(* CODESYS project railCtrl1023.project

Project tree, tasks and I/O mapping:
  Device : CODESYS SoftMotion Win V3, 3S - Smart Software Solutions GmbH, order no. 309021, version 3.5.10.0
    application Application
      libraries: Standard, * (System); VisuDialogs, * (System)
      task MainTask (cyclic, interval 4 ms, priority 1) calls PLC_PRG, floorRailInterface, yysInterface
      task VISU_TASK (cyclic, interval 100 ms, priority 31) calls VisuElems.Visu_Prg
      program PLC_PRG [ST]
      floor_rail/
        program floorRailInterface [ST]: floorRailInterface_Status, floorRailInterface_Cmd
        struct_floor_rail/
          data type OilBlockUnit_Base
          data type OilBlockUnit_Status
          data type OilBlockUnit_Cmd
          data type OilBlockUnit_Status_Loc
          data type OilBlockUnit_Status_PosVal
          data type RatioValveD1
          data type RatioValveD2
          data type RatioValveD4
          data type RatioValveD3
          data type RatioValveD5
          data type RatioValveD6
          data type RatioValveD7
          UICell/
            data type UICell_OilBlock_Info
            data type UICell_OilBlock_Button
            data type UICell_RVD3
            data type UICell_RVD1
            data type UICell_RVD2
            data type UICell_RVD5
            data type UICell_RVD4
            data type UICell_RVD6
            data type UICell_RVD7
            data type UICell_OilBlock_Module
            data type UICell_OilBlock_Module_Info
            data type UICell_OilBlock_Module_Button
          data type propValve_Struct
        text list TextList
      ceiling_rail/
        struct_ceiling_rail/
      yy_station/
        struct_yystation/
          data type YyStation_Cmd
          data type YyStation_Status
          data type YyStation
        program yysInterface [ST]: yysInterface_Status, yysInterface_Cmd
      can/
        function swmc_C00_Rx [ST]
        struct_can/
          data type Can_baseframe
          data type Can_BUS_8Inputs
          data type Can_BUS_8Outputs
          data type Can_Bus_RXMsg_Buff
          data type Can_Bus_TXMsg_Buff
        function swmc_C00_Tx [ST]
        function CAN_Send_Data_SWMC [ST]
        function swmc_C01_Rx [ST]
        function swmc_C01_Tx [ST]
        function swmc_C02_Rx [ST]
        function swmc_C02_Tx [ST]
        function swmc_C09_Rx [ST]
        function swmc_C10_Rx [ST]
      global variables gImple
      global variables gUI
      global variables gCan
      display/
        visualisation YY_Station_Display
        Orig/
          visualisation Floor_Rail1
          Module/
            visualisation OilBlock_PrimButton
            visualisation OilBlock_PrimInfo
            visualisation ModuleX2
            visualisation ModuleX1
            visualisation ModuleX3
            visualisation ModuleX8
            visualisation ModuleX4
            visualisation ModuleX5
            visualisation ModuleDTD
          visualisation Floor_Rail2
          visualisation Floor_Rail_345
          visualisation Floor_Rail6
          visualisation Floor_Rail7
          visualisation Floor_Rail_12
        visualisation Floor_Rail
        visualisation main_UI
    SoftMotion General Axis Pool
  libraries: VisuSymbols, 3.5.10.0 (System)
  text list GlobalTextList
*)

// Device/Application/yy_station/struct_yystation/YyStation_Cmd
TYPE YyStation_Cmd :
STRUCT
	InverterFan_Ctrl  		:BOOL;   //变频风机控制 0x400-1.0
	OilPumpFan_Ctrl   		:BOOL;   //油泵风机控制 0x400-1.1
	//------以下变量暂未使用,取自水平库-----------------------------------
	OilPumpMotor_Ctrl 		:BOOL;   //油泵电机控制
	OilPumpMotor_PN_Ctrl 	:BOOL;   //油泵电机正反转控制
	HL_Mode_Ctrl 			:BOOL;   //高低速模式
	KEEP_Mode_Ctrl          :BOOL;   //恒速模式
	Energy_Swith			:BOOL;   //储能控制
	Oil_Pre_Val             :WORD;   //油压控制
END_STRUCT
END_TYPE

// Device/Application/yy_station/struct_yystation/YyStation_Status
TYPE YyStation_Status :
STRUCT

	pressureStatus					: REAL;		//压力开关S1|0x300-Byt1~2
	temperatureStatus				: REAL;		//温度开关S14|0x300-Byt3~4
	yeweiStatus						: BOOL;		//液位开关S15|0x300-Byt5~6

	FrequencyConversion_Fault 		: BOOL;			//变频故障|0x300-7.0
	FrequencyConversion_Run 		: BOOL;			//变频运行|0x300-7.1
	HydraulicStation_Power			: BOOL;			//液压站上电-状态|0x300-7.2
	Control_Power					: BOOL;			//控制总电源上电状态|0x300-7.3
	InverterFan_Run 				: BOOL;			//变频风机运行状态|0x300-7.4
	OilPumpFan						: BOOL;			//冷却油泵状态|0x300-7.5
	OilPumpM_Fault 					: BOOL;			//油泵电机故障状态|0x300-7.6
	InverterFan_Fault 				: BOOL;			//变频风机故障|0x300-7.7
	
	//地轨部分压力传感器
	pressureV2						: REAL;			//压力传感器S2P|0x316-Byt1~2
	pressureV3						: REAL;			//压力传感器S3P|0x316-Byt3~4
	pressureV4						: REAL;			//压力传感器S4P|0x326-Byt1~2
	pressureV5						: REAL;			//压力传感器S5P|0x326-Byt3~4
	//天轨部分压力传感器
	pressureV8						: REAL;			//压力传感器S8P|0x356-Byt1~2
	pressureV9						: REAL;			//压力传感器S9P|0x356-Byt3~4
	pressureV10						: REAL;			//压力传感器S10P|0x366-Byt1~2
	pressureV11						: REAL;			//压力传感器S11P|0x366-Byt3~4
	

	

END_STRUCT
END_TYPE

// Device/Application/yy_station/struct_yystation/YyStation
TYPE YyStation :
STRUCT
	Cmd		:YyStation_Cmd;		//液压站指令
	Status	:YyStation_Status;	//液压站状态
	
END_STRUCT
END_TYPE

// Device/Application/can/struct_can/Can_baseframe
TYPE Can_baseframe :
STRUCT
	id		: UINT;
	data	: ARRAY[1..8] OF BYTE;
END_STRUCT
END_TYPE

// Device/Application/can/struct_can/Can_BUS_8Inputs
TYPE Can_BUS_8Inputs :          //输入缓存结构 EL6751-8Message_IN
STRUCT
	TxCounter			: UINT;
	RxCounter			: UINT;
	NoOfRxMessages 	 	: UINT;
	TransactionNumber	: UINT;
	RXMsg				: ARRAY[1..8] OF Can_Bus_RXMsg_Buff;
	CAN_State			: UINT;
	Align				: UINT;
	RX_Error_Cnt		: BYTE;
	TX_Error_Cnt		: BYTE;
END_STRUCT
END_TYPE

// Device/Application/can/struct_can/Can_BUS_8Outputs
TYPE Can_BUS_8Outputs :		//输出缓存结构 EL6751-8Message_OUT
STRUCT
	TxCounter		: UINT;
	RxCounter		: UINT;
	NoOfTxMessages 	: UINT;
	TXMsg			: ARRAY[1..8] OF Can_Bus_TXMsg_Buff;
	CAN_Control		: UINT;
END_STRUCT
END_TYPE

// Device/Application/can/struct_can/Can_Bus_RXMsg_Buff
TYPE Can_Bus_RXMsg_Buff:
STRUCT
	RxMsg_CobId		: UINT;
	RxMsg_Byte  	: ARRAY[1..8] OF BYTE;
END_STRUCT
END_TYPE

// Device/Application/can/struct_can/Can_Bus_TXMsg_Buff
TYPE Can_Bus_TXMsg_Buff :
STRUCT
	TxMsg_TransactionNumber		: UINT;
	TxMsg_CobId					: UINT;
	TxMsg_Byte  				: ARRAY[1..8] OF BYTE;
END_STRUCT
END_TYPE

// Device/Application/floor_rail/struct_floor_rail/OilBlockUnit_Base
TYPE OilBlockUnit_Base :
STRUCT
	cmd		:OilBlockUnit_Cmd;				//发送油缸指令
	status	:OilBlockUnit_Status;			//油缸状态
	cnt     :UINT;			  				//超时计数

END_STRUCT
END_TYPE

// Device/Application/floor_rail/struct_floor_rail/OilBlockUnit_Status
TYPE OilBlockUnit_Status :
STRUCT
	
	posVal			:OilBlockUnit_Status_PosVal;	//传感器位置值
	locStat			:OilBlockUnit_Status_Loc;		//位置状态
	
END_STRUCT
END_TYPE

// Device/Application/floor_rail/struct_floor_rail/OilBlockUnit_Cmd
TYPE OilBlockUnit_Cmd :
STRUCT
	E_Open	:BOOL;
	R_Open 	:BOOL;
END_STRUCT
END_TYPE

// Device/Application/floor_rail/struct_floor_rail/OilBlockUnit_Status_Loc
{attribute 'qualified_only'}
{attribute 'strict'}
TYPE OilBlockUnit_Status_Loc :
(
	enum_Run  		:= 0,   //运行中
	enum_Extend 	:= 1,	//伸出完成
	enum_Retract  	:= 2,	//缩回完成

	enum_Err  		:= 10   //错误
);
END_TYPE

// Device/Application/floor_rail/struct_floor_rail/OilBlockUnit_Status_PosVal
TYPE OilBlockUnit_Status_PosVal :
STRUCT
	Extend 		:REAL;    //伸出位置
	Retract   	:REAL;    //收回位置
	Current 	:REAL;    //当前位置
END_STRUCT
END_TYPE

// Device/Application/floor_rail/struct_floor_rail/RatioValveD1
TYPE RatioValveD1 :
STRUCT
	percenVal	: WORD;              				//比例阀DTD1|0x410-Byt1~2 0-65535 对应 0-100
	
	RVD1		:ARRAY[1..12] OF OilBlockUnit_Base;
	
	D00Q1	 	: OilBlockUnit_Base;				//DTD1连接的油缸
	D00Q2	 	: OilBlockUnit_Base;				//DTD1连接的油缸
	
	D28L1	 	: OilBlockUnit_Base;				//DTD1连接的油缸
	D28L2	 	: OilBlockUnit_Base;				//DTD1连接的油缸
	
	D29L	 	: OilBlockUnit_Base;				//DTD1连接的油缸
	D30L	 	: OilBlockUnit_Base;				//DTD1连接的油缸	

	D00L1	 	: OilBlockUnit_Base;				//DTD1连接的油缸
	D00L2	 	: OilBlockUnit_Base;				//DTD1连接的油缸
	
	D01L	 	: OilBlockUnit_Base;				//DTD1连接的油缸
	
	D28Q	 	: OilBlockUnit_Base;				//DTD1连接的油缸
	D29Q	 	: OilBlockUnit_Base;				//DTD1连接的油缸
		
	D30Q	 	: OilBlockUnit_Base;				//DTD1连接的油缸
	
	END_STRUCT
END_TYPE

// Device/Application/floor_rail/struct_floor_rail/RatioValveD2
TYPE RatioValveD2 :
STRUCT
	percenVal	: WORD;              				//比例阀DTD2|0x410-Byt3~4 0-65535 对应 0-100
	
	RVD2		:ARRAY[1..11] OF OilBlockUnit_Base;
	
	D02L	 	: OilBlockUnit_Base;				//DTD2连接的油缸
	D03L	 	: OilBlockUnit_Base;				//DTD2连接的油缸
	D04L	 	: OilBlockUnit_Base;				//DTD2连接的油缸
	
	D05L	 	: OilBlockUnit_Base;				//DTD2连接的油缸
	
	D06L	 	: OilBlockUnit_Base;				//DTD2连接的油缸
	D07L	 	: OilBlockUnit_Base;				//DTD2连接的油缸
	D08L	 	: OilBlockUnit_Base;				//DTD2连接的油缸
	
	D09L	 	: OilBlockUnit_Base;				//DTD2连接的油缸
	
	D10L	 	: OilBlockUnit_Base;				//DTD2连接的油缸
	D11L	 	: OilBlockUnit_Base;				//DTD2连接的油缸
	D12L	 	: OilBlockUnit_Base;				//DTD2连接的油缸

END_STRUCT
END_TYPE

// Device/Application/floor_rail/struct_floor_rail/RatioValveD4
TYPE RatioValveD4 :
STRUCT
	percenVal	: WORD;              				//比例阀DTD3|0x410-Byt5~6 0-65535 对应 0-100
	
	RVD4		:ARRAY[1..8] OF OilBlockUnit_Base;
	
	D05Q1	 	: OilBlockUnit_Base;				//DTD3连接的油缸
	D05Q2	 	: OilBlockUnit_Base;				//DTD3连接的油缸
	D06Q1	 	: OilBlockUnit_Base;				//DTD3连接的油缸
	D06Q2	 	: OilBlockUnit_Base;				//DTD3连接的油缸
	D07Q1	 	: OilBlockUnit_Base;				//DTD3连接的油缸
	D07Q2	 	: OilBlockUnit_Base;				//DTD3连接的油缸
	D08Q1	 	: OilBlockUnit_Base;				//DTD3连接的油缸
	D08Q2	 	: OilBlockUnit_Base;				//DTD3连接的油缸
END_STRUCT
END_TYPE

// Device/Application/floor_rail/struct_floor_rail/RatioValveD3
TYPE RatioValveD3 :
STRUCT
	percenVal	: WORD;              				//比例阀DTD4|0x410-Byt7~8 0-65535 对应 0-100
	
	RVD3		:ARRAY[1..8] OF OilBlockUnit_Base;
	
	D01Q1	 	: OilBlockUnit_Base;				//DTD4连接的油缸
	D01Q2	 	: OilBlockUnit_Base;				//DTD4连接的油缸
	D02Q1	 	: OilBlockUnit_Base;				//DTD4连接的油缸
	D02Q2	 	: OilBlockUnit_Base;				//DTD4连接的油缸	
	D03Q1	 	: OilBlockUnit_Base;				//DTD4连接的油缸
	D03Q2	 	: OilBlockUnit_Base;				//DTD4连接的油缸
	D04Q1	 	: OilBlockUnit_Base;				//DTD4连接的油缸
	D04Q2	 	: OilBlockUnit_Base;				//DTD4连接的油缸
END_STRUCT
END_TYPE

// Device/Application/floor_rail/struct_floor_rail/RatioValveD5
TYPE RatioValveD5 :
STRUCT
	percenVal	: WORD;              				//比例阀DTD5|0x411-Byt1~2 0-65535 对应 0-100
	
	RVD5		:ARRAY[1..8] OF OilBlockUnit_Base;
	
	D09Q1	 	: OilBlockUnit_Base;				//DTD5连接的油缸
	D09Q2	 	: OilBlockUnit_Base;				//DTD5连接的油缸
	D10Q1	 	: OilBlockUnit_Base;				//DTD5连接的油缸
	D10Q2	 	: OilBlockUnit_Base;				//DTD5连接的油缸
	D11Q1	 	: OilBlockUnit_Base;				//DTD5连接的油缸
	D11Q2	 	: OilBlockUnit_Base;				//DTD5连接的油缸	
	D12Q1	 	: OilBlockUnit_Base;				//DTD5连接的油缸
	D12Q2	 	: OilBlockUnit_Base;				//DTD5连接的油缸
END_STRUCT
END_TYPE

// Device/Application/floor_rail/struct_floor_rail/RatioValveD6
TYPE RatioValveD6 :
STRUCT
	percenVal	: WORD;              				//比例阀DTD6|0x420-Byt1~2 0-65535 对应 0-100
	
	RVD6		:ARRAY[1..8] OF OilBlockUnit_Base;
	
	D13Q	 	: OilBlockUnit_Base;				//DTD6连接的油缸
	D13L	 	: OilBlockUnit_Base;				//DTD6连接的油缸
	D14Q	 	: OilBlockUnit_Base;				//DTD6连接的油缸
	D14L	 	: OilBlockUnit_Base;				//DTD6连接的油缸
	D15Q	 	: OilBlockUnit_Base;				//DTD6连接的油缸
	D15L	 	: OilBlockUnit_Base;				//DTD6连接的油缸
	D16L1	 	: OilBlockUnit_Base;				//DTD6连接的油缸
	D16L2	 	: OilBlockUnit_Base;				//DTD6连接的油缸

END_STRUCT
END_TYPE

// Device/Application/floor_rail/struct_floor_rail/RatioValveD7
TYPE RatioValveD7 :
STRUCT
	percenVal	: WORD;              				//比例阀DTD7|0x420-Byt3~4 0-65535 对应 0-100
	
	RVD7		:ARRAY[1..23] OF OilBlockUnit_Base;
	
	D17Q	 	: OilBlockUnit_Base;				//DTD7连接的油缸
	D17L1	 	: OilBlockUnit_Base;				//DTD7连接的油缸
	D17L2	 	: OilBlockUnit_Base;				//DTD7连接的油缸
	D18Q	 	: OilBlockUnit_Base;				//DTD7连接的油缸
	D18L	 	: OilBlockUnit_Base;				//DTD7连接的油缸
	D19Q	 	: OilBlockUnit_Base;				//DTD7连接的油缸
	D19L	 	: OilBlockUnit_Base;				//DTD7连接的油缸
	D20Q	 	: OilBlockUnit_Base;				//DTD7连接的油缸
	D20L	 	: OilBlockUnit_Base;				//DTD7连接的油缸
	D21Q	 	: OilBlockUnit_Base;				//DTD7连接的油缸
	D21L	 	: OilBlockUnit_Base;				//DTD7连接的油缸
	D22Q	 	: OilBlockUnit_Base;				//DTD7连接的油缸
	D22L	 	: OilBlockUnit_Base;				//DTD7连接的油缸
	D23Q	 	: OilBlockUnit_Base;				//DTD7连接的油缸
	D23L	 	: OilBlockUnit_Base;				//DTD7连接的油缸
	D24Q	 	: OilBlockUnit_Base;				//DTD7连接的油缸
	D24L	 	: OilBlockUnit_Base;				//DTD7连接的油缸
	D25Q	 	: OilBlockUnit_Base;				//DTD7连接的油缸
	D25L	 	: OilBlockUnit_Base;				//DTD7连接的油缸
	D26Q	 	: OilBlockUnit_Base;				//DTD7连接的油缸
	D26L	 	: OilBlockUnit_Base;				//DTD7连接的油缸
	D27L1	 	: OilBlockUnit_Base;				//DTD7连接的油缸
	D27L2	 	: OilBlockUnit_Base;				//DTD7连接的油缸



END_STRUCT
END_TYPE

// Device/Application/floor_rail/struct_floor_rail/UICell/UICell_OilBlock_Info
TYPE UICell_OilBlock_Info :
STRUCT
	strName			:STRING;
	rPosition		:REAL;
	rPercent		:REAL;
END_STRUCT
END_TYPE

// Device/Application/floor_rail/struct_floor_rail/UICell/UICell_OilBlock_Button
TYPE UICell_OilBlock_Button :
STRUCT
	bExtend			: BOOL;	
	bRetract		: BOOL;
	bStop			: BOOL;
END_STRUCT
END_TYPE

// Device/Application/floor_rail/struct_floor_rail/UICell/UICell_RVD3
TYPE UICell_RVD3 :
STRUCT
	bRVD3_enable	:BOOL;
	rRVD3Percent	:REAL;
	S1		:UICell_OilBlock_Button;
	D01Q1	:UICell_OilBlock_Info;
	D01Q2	:UICell_OilBlock_Info;
	D02Q1	:UICell_OilBlock_Info;
	D02Q2	:UICell_OilBlock_Info;
	
	D03Q1	:UICell_OilBlock_Info;
	D03Q2	:UICell_OilBlock_Info;
	D04Q1	:UICell_OilBlock_Info;
	D04Q2	:UICell_OilBlock_Info;

END_STRUCT
END_TYPE

// Device/Application/floor_rail/struct_floor_rail/UICell/UICell_RVD1
TYPE UICell_RVD1 :
STRUCT
	
	bRVD1_enable	:BOOL;
	rRVD1Percent	:REAL;

	S1		:UICell_OilBlock_Button;
	D00Q1	:UICell_OilBlock_Info;
	D00Q2	:UICell_OilBlock_Info;
	
	
	S2		:UICell_OilBlock_Button;
	D28L1	:UICell_OilBlock_Info;
	D28L2	:UICell_OilBlock_Info;
	
	S3		:UICell_OilBlock_Button;
	D29L	:UICell_OilBlock_Info;
	D30L	:UICell_OilBlock_Info;
	
	S4		:UICell_OilBlock_Button;
	D00L1	:UICell_OilBlock_Info;
	D00L2	:UICell_OilBlock_Info;
	
	S5		:UICell_OilBlock_Button;
	D01L	:UICell_OilBlock_Info;

	S6		:UICell_OilBlock_Button;
	D28Q	:UICell_OilBlock_Info;
	D29Q	:UICell_OilBlock_Info;
	
	S7		:UICell_OilBlock_Button;
	D30Q	:UICell_OilBlock_Info;

END_STRUCT
END_TYPE

// Device/Application/floor_rail/struct_floor_rail/UICell/UICell_RVD2
TYPE UICell_RVD2 :
STRUCT
	
	bRVD2_enable	:BOOL;
	rRVD2Percent	:REAL;
	
	S1		:UICell_OilBlock_Button;
	D02L	:UICell_OilBlock_Info;
	D03L	:UICell_OilBlock_Info;
	D04L	:UICell_OilBlock_Info;
	
	S2		:UICell_OilBlock_Button;
	D05L	:UICell_OilBlock_Info;
	
	S3		:UICell_OilBlock_Button;
	D06L	:UICell_OilBlock_Info;
	D07L	:UICell_OilBlock_Info;
	D08L	:UICell_OilBlock_Info;
	
	S4		:UICell_OilBlock_Button;
	D09L	:UICell_OilBlock_Info;

	S5		:UICell_OilBlock_Button;
	D10L	:UICell_OilBlock_Info;
	D11L	:UICell_OilBlock_Info;
	D12L	:UICell_OilBlock_Info;

END_STRUCT
END_TYPE

// Device/Application/floor_rail/struct_floor_rail/UICell/UICell_RVD5
TYPE UICell_RVD5 :
STRUCT
	bRVD5_enable	:BOOL;
	rRVD5Percent	:REAL;
	S1		:UICell_OilBlock_Button;
	D09Q1	:UICell_OilBlock_Info;
	D09Q2	:UICell_OilBlock_Info;
	D10Q1	:UICell_OilBlock_Info;
	D10Q2	:UICell_OilBlock_Info;
	
	D11Q1	:UICell_OilBlock_Info;
	D11Q2	:UICell_OilBlock_Info;
	D12Q1	:UICell_OilBlock_Info;
	D12Q2	:UICell_OilBlock_Info;

END_STRUCT
END_TYPE

// Device/Application/floor_rail/struct_floor_rail/UICell/UICell_RVD4
TYPE UICell_RVD4 :
STRUCT
	bRVD4_enable	:BOOL;
	rRVD4Percent	:REAL;
	S1		:UICell_OilBlock_Button;
	D05Q1	:UICell_OilBlock_Info;
	D05Q2	:UICell_OilBlock_Info;
	D06Q1	:UICell_OilBlock_Info;
	D06Q2	:UICell_OilBlock_Info;

	D07Q1	:UICell_OilBlock_Info;
	D07Q2	:UICell_OilBlock_Info;
	D08Q1	:UICell_OilBlock_Info;
	D08Q2	:UICell_OilBlock_Info;

END_STRUCT
END_TYPE

// Device/Application/floor_rail/struct_floor_rail/UICell/UICell_RVD6
TYPE UICell_RVD6 :
STRUCT
	bRVD6_enable	:BOOL;
	rRVD6Percent	:REAL;
	S1		:UICell_OilBlock_Button;
	D13Q	:UICell_OilBlock_Info;
	D14Q	:UICell_OilBlock_Info;
		
	S2		:UICell_OilBlock_Button;
	D15Q	:UICell_OilBlock_Info;
	
	S3		:UICell_OilBlock_Button;
	D13L	:UICell_OilBlock_Info;
	D14L	:UICell_OilBlock_Info;
	
	S4		:UICell_OilBlock_Button;
	D15L	:UICell_OilBlock_Info;

	S5		:UICell_OilBlock_Button;
	D16L1	:UICell_OilBlock_Info;
	D16L2	:UICell_OilBlock_Info;


END_STRUCT
END_TYPE

// Device/Application/floor_rail/struct_floor_rail/UICell/UICell_RVD7
TYPE UICell_RVD7 :
STRUCT
	bRVD7_enable	:BOOL;
	rRVD7Percent	:REAL;
	
	S1		:UICell_OilBlock_Button;
	D18L	:UICell_OilBlock_Info;
	D19L	:UICell_OilBlock_Info;
	D20L	:UICell_OilBlock_Info;
	D21L	:UICell_OilBlock_Info;
		
	S2		:UICell_OilBlock_Button;
	D22L	:UICell_OilBlock_Info;
	
	S3		:UICell_OilBlock_Button;
	D23L	:UICell_OilBlock_Info;
	D24L	:UICell_OilBlock_Info;
	D25L	:UICell_OilBlock_Info;
	D26L	:UICell_OilBlock_Info;
	
	S4		:UICell_OilBlock_Button;
	D17Q	:UICell_OilBlock_Info;
	D18Q	:UICell_OilBlock_Info;
	D19Q	:UICell_OilBlock_Info;
	D20Q	:UICell_OilBlock_Info;
	D21Q	:UICell_OilBlock_Info;

	S5		:UICell_OilBlock_Button;
	D22Q	:UICell_OilBlock_Info;
	D23Q	:UICell_OilBlock_Info;
	D24Q	:UICell_OilBlock_Info;
	D25Q	:UICell_OilBlock_Info;
	D26Q	:UICell_OilBlock_Info;
	
	S6		:UICell_OilBlock_Button;
	D17L1	:UICell_OilBlock_Info;
	D17L2	:UICell_OilBlock_Info;
	
	S7		:UICell_OilBlock_Button;
	D27L1	:UICell_OilBlock_Info;
	D27L2	:UICell_OilBlock_Info;

END_STRUCT
END_TYPE

// Device/Application/floor_rail/struct_floor_rail/propValve_Struct
TYPE propValve_Struct :
STRUCT
	D1	:RatioValveD1;
	D2	:RatioValveD2;
	D3	:RatioValveD3;
	D4	:RatioValveD4;
	D5	:RatioValveD5;
	D6	:RatioValveD6;
	D7	:RatioValveD7;

	
END_STRUCT
END_TYPE

// Device/Application/floor_rail/struct_floor_rail/UICell/UICell_OilBlock_Module
TYPE UICell_OilBlock_Module :
STRUCT
	
	sColumn				:ARRAY[1..8] OF UICell_OilBlock_Module_Button;
	sRow				:ARRAY[1..8] OF UICell_OilBlock_Module_Info;

END_STRUCT
END_TYPE

// Device/Application/floor_rail/struct_floor_rail/UICell/UICell_OilBlock_Module_Info
TYPE UICell_OilBlock_Module_Info :
STRUCT
	strName			:STRING;
	rPosition		:REAL;
	rPercent		:REAL;
END_STRUCT
END_TYPE

// Device/Application/floor_rail/struct_floor_rail/UICell/UICell_OilBlock_Module_Button
TYPE UICell_OilBlock_Module_Button :
STRUCT
	bExtend			: BOOL;	
	bRetract		: BOOL;
	bStop			: BOOL;
END_STRUCT
END_TYPE

// Device/Application/gImple
{attribute 'qualified_only'}
VAR_GLOBAL
	





	hydraPresStation	:YyStation;
	propValve			:propValve_Struct;
	
	
	
END_VAR

// Device/Application/gUI
{attribute 'qualified_only'}
VAR_GLOBAL
	
//液压站部分
	//压力
	rPressureVal1				:REAL;			//压力传感器SQ1P(压力开关S1)
	rPressureVal2				:REAL;			//压力传感器SQ2P
	rPressureVal3				:REAL;			//压力传感器SQ3P
	rPressureVal4				:REAL;			//压力传感器SQ4P
	rPressureVal5				:REAL;			//压力传感器SQ5P	
	//状态
	rTemperature				:REAL;			//温度值
	bFluidLevel					:BOOL;			//液位值
	
	bYysPower	 		 		:BOOL;			//液压站上电
	bCtrlPower	  		 		:BOOL;			//控制电源上电
	bFreqConverterFan			:BOOL;    	    //变频风机启动
	bFreqConverter				:BOOL;			//变频器运行
	
	bOilPumpM_Fault				:BOOL;			//油泵电机故障
	bOilPumpFan					:BOOL;			//油泵冷却风机  无故障
	bFreqConverter_Fault		:BOOL;			//变频器故障
	bFreqConverterFan_Fault		:BOOL;			//变频器风机故障
	//控制指令
	cmdInverterFan				:BOOL;			//变频风机控制
	cmdOilPumpFan				:BOOL;    	    //油泵风机控制
	cmdOilPumpM					:BOOL;			//油泵电机控制
	cmdOilPrePercent			:REAL;			//油压控制百分比
	cmdOilPre_EN				:BOOL;			//油压使能

	//DTD01
	DiG1						:UICell_RVD1;
	DiG2						:UICell_RVD2;
	DiG3						:UICell_RVD3;
	DiG4						:UICell_RVD4;
	DiG5						:UICell_RVD5;
	DiG6						:UICell_RVD6;
	DiG7						:UICell_RVD7;
	
END_VAR

// Device/Application/gCan
{attribute 'qualified_only'}
VAR_GLOBAL
	//SWMC
	C0TxMsg			AT%QW50:Can_BUS_8Outputs;	
	C0RxMsg			AT%IW50:Can_BUS_8Inputs;
	C0RxCounter			   : UINT;
	
	C1TxMsg			AT%QW51:Can_BUS_8Outputs;	
	C1RxMsg			AT%IW51:Can_BUS_8Inputs;
	C1RxCounter			   : UINT;
	
	C2TxMsg			AT%QW52:Can_BUS_8Outputs;	
	C2RxMsg			AT%IW52:Can_BUS_8Inputs;
	C2RxCounter			   : UINT;

	C9TxMsg			AT%QW55:Can_BUS_8Outputs;	
	C9RxMsg			AT%IW55:Can_BUS_8Inputs;
	C9RxCounter			   : UINT;
	
	C10TxMsg		AT%QW56:Can_BUS_8Outputs;	
	C10RxMsg		AT%IW56:Can_BUS_8Inputs;
	C10RxCounter		   : UINT;
	
	
	
	
	
	
	C5TxMsg			AT%QW53:Can_BUS_8Outputs;	
	C5RxMsg			AT%IW53:Can_BUS_8Inputs;
	C5RxCounter			   : UINT;
	
	C6TxMsg			AT%QW54:Can_BUS_8Outputs;	
	C6RxMsg			AT%IW54:Can_BUS_8Inputs;
	C6RxCounter			   : UINT;
	
	
	C11TxMsg		AT%QW57:Can_BUS_8Outputs;	
	C11RxMsg		AT%IW57:Can_BUS_8Inputs;
	C11RxCounter		   : UINT;
	
	C12TxMsg		AT%QW58:Can_BUS_8Outputs;	
	C12RxMsg		AT%IW58:Can_BUS_8Inputs;
	C12RxCounter		   : UINT;	
END_VAR

// Device/Application/PLC_PRG
PROGRAM PLC_PRG
VAR
END_VAR

END_PROGRAM

// Device/Application/floor_rail/floorRailInterface
PROGRAM floorRailInterface
VAR
	
END_VAR

floorRailInterface_Status();

ACTION floorRailInterface_Status:
//比例阀DTD1
gUI.DiG1.D00Q1.rPosition:=gImple.propValve.D1.D00Q1.status.posVal.Current;
gUI.DiG1.D00Q2.rPosition:=gImple.propValve.D1.D00Q2.status.posVal.Current;
gUI.DiG1.D28L1.rPosition:=gImple.propValve.D1.D28L1.status.posVal.Current;
gUI.DiG1.D28L2.rPosition:=gImple.propValve.D1.D28L2.status.posVal.Current;
gUI.DiG1.D29L.rPosition	:=gImple.propValve.D1.D29L.status.posVal.Current;
gUI.DiG1.D30L.rPosition	:=gImple.propValve.D1.D30L.status.posVal.Current;
gUI.DiG1.D00L1.rPosition:=gImple.propValve.D1.D00L1.status.posVal.Current;
gUI.DiG1.D00L2.rPosition:=gImple.propValve.D1.D00L2.status.posVal.Current;
gUI.DiG1.D01L.rPosition	:=gImple.propValve.D1.D01L.status.posVal.Current;
gUI.DiG1.D28Q.rPosition	:=gImple.propValve.D1.D28Q.status.posVal.Current;
gUI.DiG1.D29Q.rPosition	:=gImple.propValve.D1.D29Q.status.posVal.Current;
gUI.DiG1.D30Q.rPosition	:=gImple.propValve.D1.D30Q.status.posVal.Current;

gUI.DiG2.D02L.rPosition	:=gImple.propValve.D2.D02L.status.posVal.Current;
gUI.DiG2.D03L.rPosition	:=gImple.propValve.D2.D03L.status.posVal.Current;
gUI.DiG2.D04L.rPosition	:=gImple.propValve.D2.D04L.status.posVal.Current;
gUI.DiG2.D05L.rPosition	:=gImple.propValve.D2.D05L.status.posVal.Current;
gUI.DiG2.D06L.rPosition	:=gImple.propValve.D2.D06L.status.posVal.Current;
gUI.DiG2.D07L.rPosition	:=gImple.propValve.D2.D07L.status.posVal.Current;
gUI.DiG2.D08L.rPosition	:=gImple.propValve.D2.D08L.status.posVal.Current;
gUI.DiG2.D09L.rPosition	:=gImple.propValve.D2.D09L.status.posVal.Current;

gUI.DiG3.D01Q1.rPosition	:=gImple.propValve.D3.D01Q1.status.posVal.Current;
gUI.DiG3.D01Q2.rPosition	:=gImple.propValve.D3.D01Q2.status.posVal.Current;
gUI.DiG3.D02Q1.rPosition	:=gImple.propValve.D3.D02Q1.status.posVal.Current;
gUI.DiG3.D02Q2.rPosition	:=gImple.propValve.D3.D02Q2.status.posVal.Current;
gUI.DiG3.D03Q1.rPosition	:=gImple.propValve.D3.D03Q1.status.posVal.Current;
gUI.DiG3.D03Q2.rPosition	:=gImple.propValve.D3.D03Q2.status.posVal.Current;
gUI.DiG3.D04Q1.rPosition	:=gImple.propValve.D3.D04Q1.status.posVal.Current;
gUI.DiG3.D04Q2.rPosition	:=gImple.propValve.D3.D04Q2.status.posVal.Current;
gUI.DiG4.D05Q1.rPosition	:=gImple.propValve.D4.D05Q1.status.posVal.Current;
gUI.DiG4.D05Q2.rPosition	:=gImple.propValve.D4.D05Q2.status.posVal.Current;
gUI.DiG4.D06Q1.rPosition	:=gImple.propValve.D4.D06Q1.status.posVal.Current;
gUI.DiG4.D06Q2.rPosition	:=gImple.propValve.D4.D06Q2.status.posVal.Current;
gUI.DiG4.D07Q1.rPosition	:=gImple.propValve.D4.D07Q1.status.posVal.Current;
gUI.DiG4.D07Q2.rPosition	:=gImple.propValve.D4.D07Q2.status.posVal.Current;
gUI.DiG4.D08Q1.rPosition	:=gImple.propValve.D4.D08Q1.status.posVal.Current;
gUI.DiG4.D08Q2.rPosition	:=gImple.propValve.D4.D08Q2.status.posVal.Current;
gUI.DiG5.D09Q1.rPosition	:=gImple.propValve.D5.D09Q1.status.posVal.Current;
gUI.DiG5.D09Q2.rPosition	:=gImple.propValve.D5.D09Q2.status.posVal.Current;
gUI.DiG5.D10Q1.rPosition	:=gImple.propValve.D5.D10Q1.status.posVal.Current;
gUI.DiG5.D10Q2.rPosition	:=gImple.propValve.D5.D10Q2.status.posVal.Current;
gUI.DiG5.D11Q1.rPosition	:=gImple.propValve.D5.D11Q1.status.posVal.Current;
gUI.DiG5.D11Q2.rPosition	:=gImple.propValve.D5.D11Q2.status.posVal.Current;
gUI.DiG5.D12Q1.rPosition	:=gImple.propValve.D5.D12Q1.status.posVal.Current;
gUI.DiG5.D12Q2.rPosition	:=gImple.propValve.D5.D12Q2.status.posVal.Current;




gUI.DiG1.D00Q1.strName	:='D00Q1';
gUI.DiG1.D00Q2.strName	:='D00Q2';
gUI.DiG1.D28L1.strName	:='D28L1';
gUI.DiG1.D28L2.strName	:='D28L2';
gUI.DiG1.D29L.strName	:='D29L';
gUI.DiG1.D30L.strName	:='D30L';
gUI.DiG1.D00L1.strName	:='D00L1';
gUI.DiG1.D00L2.strName	:='D00L2';
gUI.DiG1.D01L.strName	:='D01L';
gUI.DiG1.D28Q.strName	:='D28Q';
gUI.DiG1.D29Q.strName	:='D29Q';
gUI.DiG1.D30Q.strName	:='D30Q';

//percentBar
(*

gUI.DiG1.D00Q1.rPercent	:=
gUI.DiG1.D00Q2.rPercent	:=
gUI.DiG1.D28L1.rPercent	:=
gUI.DiG1.D28L2.rPercent	:=
gUI.DiG1.D29L.rPercent	:=
gUI.DiG1.D30L.rPercent	:=
gUI.DiG1.D00L1.rPercent	:=
gUI.DiG1.D00L2.rPercent	:=
gUI.DiG1.D01L.rPercent	:=
gUI.DiG1.D28Q.rPercent	:=
gUI.DiG1.D29Q.rPercent	:=
gUI.DiG1.D30Q.rPercent	:=
*)
END_ACTION

METHOD floorRailInterface_Cmd : BOOL
VAR_INPUT
	pstPValve			:POINTER TO propValve_Struct;
	
END_VAR
(*
IF gUI.DiG1.bRVD1_enable THEN
	gImple.propValve.D1.percenVal:=REAL_TO_WORD(gUI.DiG1.rRVD1Percent);
ELSE
	gImple.propValve.D1.percenVal:=0;
END_IF
*)
END_METHOD

END_PROGRAM

// Device/Application/yy_station/yysInterface
PROGRAM yysInterface
VAR
	
END_VAR

yysInterface_Status();

yysInterface_Cmd
(
	ADR(gImple.hydraPresStation),		//液压站地址
	gUI.cmdInverterFan,					//变频器风机
	gUI.cmdOilPumpFan,					//油泵风机
	gUI.cmdOilPumpM,					//油泵电机
	gUI.cmdOilPrePercent,				//油压百分比
	gUI.cmdOilPre_EN					//油压使能
);

ACTION yysInterface_Status:
	//压力
	gUI.rPressureVal1:=gImple.hydraPresStation.Status.pressureStatus;	 		//压力传感器SQ1P(压力开关S1)
	gUI.rPressureVal2:=gImple.hydraPresStation.Status.pressureV2;				//压力传感器SQ2P
	gUI.rPressureVal3:=gImple.hydraPresStation.Status.pressureV3;				//压力传感器SQ3P
	gUI.rPressureVal4:=gImple.hydraPresStation.Status.pressureV4;				//压力传感器SQ4P
	gUI.rPressureVal5:=gImple.hydraPresStation.Status.pressureV5;				//压力传感器SQ5P	
	//状态
	gUI.rTemperature:=gImple.hydraPresStation.Status.temperatureStatus;			//温度值
	gUI.bFluidLevel	:=gImple.hydraPresStation.Status.yeweiStatus;				//液位值
	
	gUI.bYysPower:=gImple.hydraPresStation.Status.HydraulicStation_Power;		//液压站上电
	gUI.bCtrlPower:=gImple.hydraPresStation.Status.Control_Power;				//控制电源上电
	gUI.bFreqConverterFan:=gImple.hydraPresStation.Status.InverterFan_Run;  	//变频风机启动
	gUI.bFreqConverter:=gImple.hydraPresStation.Status.FrequencyConversion_Run;	//变频器运行
	
	gUI.bOilPumpM_Fault:=gImple.hydraPresStation.Status.OilPumpM_Fault;			//油泵电机故障
	gUI.bOilPumpFan:=gImple.hydraPresStation.Status.OilPumpFan;					//油泵冷却风机-非故障
	gUI.bFreqConverter_Fault:=gImple.hydraPresStation.Status.FrequencyConversion_Fault;	//变频器故障
	gUI.bFreqConverterFan_Fault:=gImple.hydraPresStation.Status.InverterFan_Fault;		//变频器风机故障
END_ACTION

METHOD yysInterface_Cmd : BOOL
VAR_INPUT
	psYyz						:POINTER TO YyStation;
	cmdInverterFan				:BOOL;			//变频风机控制
	cmdOilPumpFan				:BOOL;    	    //油泵风机控制
	cmdOilPumpM					:BOOL;			//油泵电机控制
	cmdOilPrePercent			:REAL;			//油压控制
	cmdOilPre_EN				:BOOL;			//油压使能
END_VAR

VAR
	bSetCondition				:BOOL;			//温度、液位等状态要求
	wOilPrePercentTemp  		:WORD;
	wOilMaxPreVal				:WORD:=50;  	//最大限制为50
	
END_VAR

//液压站故障处理？

psYyz^.Cmd.HL_Mode_Ctrl:=0;				//高低速为0
psYyz^.Cmd.Energy_Swith:=0;				//储能开关为0
psYyz^.Cmd.OilPumpMotor_PN_Ctrl:=0;		//电机正反控制为0

//bSetCondition:=条件判定,满足后可执行以下动作
//IF bSetCondition 
//THEN

IF cmdOilPumpFan THEN					//油泵风扇控制
	psYyz^.Cmd.OilPumpFan_Ctrl:=1;
ELSE
	psYyz^.Cmd.OilPumpFan_Ctrl:=0;
END_IF

IF cmdInverterFan THEN					//变频器风扇控制
	psYyz^.Cmd.InverterFan_Ctrl:=1;
ELSE
	psYyz^.Cmd.InverterFan_Ctrl:=0;	
END_IF

IF cmdOilPumpFan THEN					//电机启动
	psYyz^.Cmd.OilPumpMotor_Ctrl:=1;
	psYyz^.Cmd.KEEP_Mode_Ctrl:=1;		//恒速模式
ELSE
	psYyz^.Cmd.OilPumpMotor_Ctrl:=0;
	psYyz^.Cmd.KEEP_Mode_Ctrl:=0;
END_IF

IF cmdOilPrePercent > wOilMaxPreVal THEN	//最大限制为 50%
	cmdOilPrePercent:=wOilMaxPreVal;
END_IF

IF cmdOilPre_EN THEN						//液压使能后才输出压力值
	wOilPrePercentTemp:=REAL_TO_WORD(cmdOilPrePercent*65535/100);
ELSE
	wOilPrePercentTemp:=0;
END_IF

psYyz^.Cmd.Oil_Pre_Val := wOilPrePercentTemp;
END_METHOD

END_PROGRAM

// Device/Application/can/swmc_C00_Rx
FUNCTION swmc_C00_Rx : BOOL
VAR_INPUT
	CNT				: UINT;
	psYyz			: POINTER TO YyStation;
END_VAR
VAR
	frame	    : Can_baseframe;
	COB_ID		: UINT;
	I			: UINT;
	Pre			: UINT;
END_VAR

IF gCan.C0RxMsg.RxCounter <>  gCan.C0RxCounter THEN    //接收到新的数据
	
	FOR  I :=1 TO  gCan.C0RxMsg.NoOfRxMessages DO
		//frame :=CAN_Read_Data_SWMC(0,I);
		COB_ID :=	frame.id;    //获取ID
		CASE  COB_ID OF     //根据ID解析协议
			//C0-0x300
			16#300:           //液压站状态数据
				psYyz^.Status.HydraulicStation_Power := frame.data[1].0;     //液压站上电 
				psYyz^.Status.Control_Power :=frame.data[1].1;				 //控制总电源上电
				psYyz^.Status.OilPumpM_Fault :=frame.data[2].0;			 //油泵电机故障
				psYyz^.Status.InverterFan_Run :=frame.data[2].1;			 //变频风机
				psYyz^.Status.InverterFan_Fault :=frame.data[3].0;			 //变频风机故障
				psYyz^.Status.OilPumpFan :=frame.data[3].1;					 //SP油泵风机故障
				psYyz^.Status.FrequencyConversion_Fault :=frame.data[4].0;   //变频故障
				psYyz^.Status.FrequencyConversion_Run :=frame.data[4].1;	 //变频运行
				
			//C0-0x301
			16#301:           //液压站状态数据
				Pre :=BYTE_TO_WORD(frame.data[1]) OR SHL(BYTE_TO_WORD(frame.data[2]),8);
	 			psYyz^.Status.pressureStatus:= 	(Pre-4000)/16000.0*400;	
				Pre :=BYTE_TO_WORD(frame.data[3]) OR SHL(BYTE_TO_WORD(frame.data[4]),8);
				
			 	//???
				psYyz^.Status.yeweiStatus				:=frame.data[5].0;
				(*
				psYyz^.Status.FrequencyConversion_Fault	:=frame.data[7].0;
				psYyz^.Status.FrequencyConversion_Run	:=frame.data[7].1;
				psYyz^.Status.HydraulicStation_Power	:=frame.data[7].2;
				psYyz^.Status.Control_Power				:=frame.data[7].3;
				psYyz^.Status.InverterFan_Run			:=frame.data[7].4;
				psYyz^.Status.OilPumpFan				:=frame.data[7].5;
				psYyz^.Status.OilPumpMotor_Fault		:=frame.data[7].6;
				psYyz^.Status.InverterFan_Fault			:=frame.data[7].7;
				*)	
		END_CASE
	END_FOR
	gCan.C0RxCounter := gCan.C0RxMsg.RxCounter ;
END_IF

END_FUNCTION

// Device/Application/can/swmc_C00_Tx
FUNCTION swmc_C00_Tx : BOOL
VAR_INPUT
	CNT				: UINT;
	psYyz			: POINTER TO YyStation;
END_VAR
VAR
	senddata	: ARRAY[1..8] OF BYTE;
	Send_cnt	: UINT;
END_VAR

//控制速度--待定
Send_cnt :=  CNT MOD 3;

CASE Send_cnt OF
	
    1:
	 //C0-0x400
	 
	senddata[1].0 :=  psYyz^.Cmd.InverterFan_Ctrl; 		// 变频风机控制
	senddata[1].1 :=  psYyz^.Cmd.OilPumpFan_Ctrl;		// 油泵风机控制
	senddata[2].0 :=  psYyz^.Cmd.OilPumpMotor_Ctrl;		// 油泵电机控制    
	senddata[2].1 :=  psYyz^.Cmd.OilPumpMotor_PN_Ctrl;  // 油泵电机正反转
	senddata[3].0 :=  psYyz^.Cmd.HL_Mode_Ctrl;          // 高低速模式
	senddata[3].1 :=  psYyz^.Cmd.KEEP_Mode_Ctrl;        // 恒速模式      
	senddata[4].0 :=  0;                     			//储能开关
	senddata[5]   :=  WORD_TO_BYTE(psYyz^.Cmd.Oil_Pre_Val);      		           
	senddata[6]   :=  WORD_TO_BYTE(SHR(psYyz^.Cmd.Oil_Pre_Val,8));    //油压控制   
	senddata[7]   :=  0;           //设置A04存储夹紧块状态
	senddata[8]   :=  0; 

	 (*
	senddata[1].0 :=  psYyz^.Cmd.InverterFan_Ctrl; 		// 变频风机控制
	senddata[1].1 :=  psYyz^.Cmd.OilPumpFan_Ctrl;		// 油泵风机控制
	senddata[2]   :=  0;  
	senddata[3]   :=  0;    
	senddata[4]	  :=  0;                     			
	senddata[5]   :=  0;      		           
	senddata[6]   :=  0; 
	senddata[7]   :=  0;           
	senddata[8]   :=  0; 
	*)
	
	//发送至C0
	CAN_Send_Data_SWMC(0, 16#400,senddata);   //发送ID 0x400到 C0

END_CASE

END_FUNCTION

// Device/Application/can/CAN_Send_Data_SWMC
FUNCTION CAN_Send_Data_SWMC : BOOL
VAR_INPUT
	SWMC_ID : UINT;
	id 		: UINT;
	data	: ARRAY[1..8] OF BYTE;
END_VAR
VAR
	
END_VAR

CASE  SWMC_ID OF
	0:
	   gCan.C0TxMsg.TXMsg[1].TxMsg_CobId 	:= 8 + 32 * id;
	   gCan.C0TxMsg.TXMsg[1].TxMsg_Byte 	:= data;
	   gCan.C0TxMsg.NoOfTxMessages 		:= 1;
	   gCan.C0TxMsg.TxCounter 				:= gCan.C0TxMsg.TxCounter +1;
	1:
	   gCan.C1TxMsg.TXMsg[1].TxMsg_CobId 	:= 8 + 32 * id;
	   gCan.C1TxMsg.TXMsg[1].TxMsg_Byte 	:= data;
	   gCan.C1TxMsg.NoOfTxMessages			:=1;
	   gCan.C1TxMsg.TxCounter 				:= gCan.C0TxMsg.TxCounter +1;
	

END_CASE

END_FUNCTION

// Device/Application/can/swmc_C01_Rx
FUNCTION swmc_C01_Rx : BOOL
VAR_INPUT
	CNT				: UINT;
	psYyz			: POINTER TO YyStation;
	psDiG3			: POINTER TO RatioValveD3;
	psDiG4			: POINTER TO RatioValveD4;
	psDiG5			: POINTER TO RatioValveD5;	
END_VAR
VAR
	frame	 	    : Can_baseframe;
	COB_ID			: UINT;
	I				: UINT;
	pos				: WORD;
	Pre				: UINT;
END_VAR

IF gCan.C1RxMsg.RxCounter <>  gCan.C1RxCounter THEN    //接收到新的数据

	FOR  I := 1 TO  gCan.C1RxMsg.NoOfRxMessages DO
		COB_ID :=	frame.id;    //获取ID
		CASE COB_ID OF     //根据ID解析协议
		
			
			//C1-0x310
			16#310:           //接收C1送来的数据
				pos := BYTE_TO_WORD(frame.data[1]) OR SHL(BYTE_TO_WORD(frame.data[2]),8);  	
				psDiG3^.D01Q1.status.posVal.Current:= pos*0.1;	//驱动插销油缸D01Q1-位移传感器	
				pos := BYTE_TO_WORD(frame.data[3]) OR SHL(BYTE_TO_WORD(frame.data[4]),8);  	
				psDiG3^.D01Q2.status.posVal.Current:= pos*0.1;	//驱动插销油缸D01Q2-位移传感器	
				pos := BYTE_TO_WORD(frame.data[5]) OR SHL(BYTE_TO_WORD(frame.data[6]),8);  	
				psDiG3^.D02Q1.status.posVal.Current:= pos*0.1;	//驱动插销油缸D02Q1-位移传感器	
				pos := BYTE_TO_WORD(frame.data[7]) OR SHL(BYTE_TO_WORD(frame.data[8]),8);  	
				psDiG3^.D02Q2.status.posVal.Current:= pos*0.1;	//驱动插销油缸D02Q2-位移传感器	
			//C1-0x311
			16#311:           //接收C1送来的数据
				pos := BYTE_TO_WORD(frame.data[1]) OR SHL(BYTE_TO_WORD(frame.data[2]),8);  	
				psDiG3^.D03Q1.status.posVal.Current:= pos*0.1;	//驱动插销油缸D03Q1-位移传感器	
				pos := BYTE_TO_WORD(frame.data[3]) OR SHL(BYTE_TO_WORD(frame.data[4]),8);  	
				psDiG3^.D03Q2.status.posVal.Current:= pos*0.1;	//驱动插销油缸D03Q2-位移传感器	
				pos := BYTE_TO_WORD(frame.data[5]) OR SHL(BYTE_TO_WORD(frame.data[6]),8);  	
				psDiG3^.D04Q1.status.posVal.Current:= pos*0.1;	//驱动插销油缸D04Q1-位移传感器	
				pos := BYTE_TO_WORD(frame.data[7]) OR SHL(BYTE_TO_WORD(frame.data[8]),8);  	
				psDiG3^.D04Q2.status.posVal.Current:= pos*0.1;	//驱动插销油缸D04Q2-位移传感器
				
		//比例阀DTD4	
			//C1-0x312
			16#312:           //接收C1送来的数据
				pos := BYTE_TO_WORD(frame.data[1]) OR SHL(BYTE_TO_WORD(frame.data[2]),8);  	
				psDiG4^.D05Q1.status.posVal.Current:= pos*0.1;	//驱动插销油缸D05Q1-位移传感器	
				pos := BYTE_TO_WORD(frame.data[3]) OR SHL(BYTE_TO_WORD(frame.data[4]),8);  	
				psDiG4^.D05Q2.status.posVal.Current:= pos*0.1;	//驱动插销油缸D05Q2-位移传感器	
				pos := BYTE_TO_WORD(frame.data[5]) OR SHL(BYTE_TO_WORD(frame.data[6]),8);  	
				psDiG4^.D06Q1.status.posVal.Current:= pos*0.1;	//驱动插销油缸D06Q1-位移传感器	
				pos := BYTE_TO_WORD(frame.data[7]) OR SHL(BYTE_TO_WORD(frame.data[8]),8);  	
				psDiG4^.D06Q2.status.posVal.Current:= pos*0.1;	//驱动插销油缸D06Q2-位移传感器	
			//C1-0x313
			16#313:           //接收C1送来的数据
				pos := BYTE_TO_WORD(frame.data[1]) OR SHL(BYTE_TO_WORD(frame.data[2]),8);  	
				psDiG4^.D07Q1.status.posVal.Current:= pos*0.1;	//驱动插销油缸D07Q1-位移传感器	
				pos := BYTE_TO_WORD(frame.data[3]) OR SHL(BYTE_TO_WORD(frame.data[4]),8);  	
				psDiG4^.D07Q2.status.posVal.Current:= pos*0.1;	//驱动插销油缸D07Q2-位移传感器	
				pos := BYTE_TO_WORD(frame.data[5]) OR SHL(BYTE_TO_WORD(frame.data[6]),8);  	
				psDiG4^.D08Q1.status.posVal.Current:= pos*0.1;	//驱动插销油缸D08Q1-位移传感器	
				pos := BYTE_TO_WORD(frame.data[7]) OR SHL(BYTE_TO_WORD(frame.data[8]),8);  	
				psDiG4^.D08Q2.status.posVal.Current:= pos*0.1;	//驱动插销油缸D08Q2-位移传感器
				
		//比例阀DTD5					
			//C1-0x314
			16#314:           //接收C1送来的数据
				pos := BYTE_TO_WORD(frame.data[1]) OR SHL(BYTE_TO_WORD(frame.data[2]),8);  	
				psDiG5^.D09Q1.status.posVal.Current:= pos*0.1;	//驱动插销油缸D09Q1-位移传感器	
				pos := BYTE_TO_WORD(frame.data[3]) OR SHL(BYTE_TO_WORD(frame.data[4]),8);  	
				psDiG5^.D09Q2.status.posVal.Current:= pos*0.1;	//驱动插销油缸D09Q2-位移传感器	
				pos := BYTE_TO_WORD(frame.data[5]) OR SHL(BYTE_TO_WORD(frame.data[6]),8);  	
				psDiG5^.D10Q1.status.posVal.Current:= pos*0.1;	//驱动插销油缸D10Q1-位移传感器	
				pos := BYTE_TO_WORD(frame.data[7]) OR SHL(BYTE_TO_WORD(frame.data[8]),8);  	
				psDiG5^.D10Q2.status.posVal.Current:= pos*0.1;	//驱动插销油缸D10Q2-位移传感器	
			//C1-0x315
			16#315:           //接收C1送来的数据
				pos := BYTE_TO_WORD(frame.data[1]) OR SHL(BYTE_TO_WORD(frame.data[2]),8);  	
				psDiG5^.D11Q1.status.posVal.Current:= pos*0.1;	//驱动插销油缸D11Q1-位移传感器	
				pos := BYTE_TO_WORD(frame.data[3]) OR SHL(BYTE_TO_WORD(frame.data[4]),8);  	
				psDiG5^.D11Q2.status.posVal.Current:= pos*0.1;	//驱动插销油缸D11Q2-位移传感器	
				pos := BYTE_TO_WORD(frame.data[5]) OR SHL(BYTE_TO_WORD(frame.data[6]),8);  	
				psDiG5^.D12Q1.status.posVal.Current:= pos*0.1;	//驱动插销油缸D12Q1-位移传感器	
				pos := BYTE_TO_WORD(frame.data[7]) OR SHL(BYTE_TO_WORD(frame.data[8]),8);  	
				psDiG5^.D12Q2.status.posVal.Current:= pos*0.1;	//驱动插销油缸D12Q2-位移传感器
			
			//C1-0x316
			16#316:           //液压站状态数据
			
				Pre :=BYTE_TO_WORD(frame.data[1]) OR SHL(BYTE_TO_WORD(frame.data[2]),8);
	 			psYyz^.Status.pressureV2:= 	(Pre-4000)/16000.0*400;	
				
			    Pre :=BYTE_TO_WORD(frame.data[3]) OR SHL(BYTE_TO_WORD(frame.data[4]),8);
	 			psYyz^.Status.pressureV3:= 	(Pre-4000)/16000.0*400;	
				
			
			
			(*
				Pre :=BYTE_TO_WORD(frame.data[1]) OR SHL(BYTE_TO_WORD(frame.data[2]),8);
	 			psYyz^.Status.pressureStatus:= 	(Pre-4000)/16000.0*400;	
				Pre :=BYTE_TO_WORD(frame.data[3]) OR SHL(BYTE_TO_WORD(frame.data[4]),8);
			 	//???
				psYyz^.Status.yeweiStatus				:=frame.data[5].0;
				
				psYyz^.Status.FrequencyConversion_Fault	:=frame.data[7].0;
				psYyz^.Status.FrequencyConversion_Run	:=frame.data[7].1;
				psYyz^.Status.HydraulicStation_Power	:=frame.data[7].2;
				psYyz^.Status.Control_Power				:=frame.data[7].3;
				psYyz^.Status.InverterFan_Run			:=frame.data[7].4;
				psYyz^.Status.OilPumpFan				:=frame.data[7].5;
				psYyz^.Status.OilPumpMotor_Fault		:=frame.data[7].6;
				psYyz^.Status.InverterFan_Fault			:=frame.data[7].7;
					*)	
		END_CASE
	END_FOR


	gCan.C0RxCounter := gCan.C0RxMsg.RxCounter ;
END_IF

END_FUNCTION

// Device/Application/can/swmc_C01_Tx
FUNCTION swmc_C01_Tx : BOOL
VAR_INPUT
	CNT				: UINT;
	psDiG1			: POINTER TO RatioValveD1;
	psDiG2			: POINTER TO RatioValveD2;		
	psDiG3			: POINTER TO RatioValveD3;
	psDiG4			: POINTER TO RatioValveD4;
	psDiG5			: POINTER TO RatioValveD5;
END_VAR
VAR
	senddata	: ARRAY[1..8] OF BYTE;
	Send_cnt	: UINT;
END_VAR

//控制速度--待定
Send_cnt :=  CNT MOD 3;

CASE Send_cnt OF
	
    1:
	 //C1-0x410
	senddata[1] :=  WORD_TO_BYTE(psDiG1^.percenVal);  		   //发送DTD1比例阀值
	senddata[2] :=  WORD_TO_BYTE(SHR(psDiG1^.percenVal,8));    //0-65535  对应0-100  
	senddata[3] :=  WORD_TO_BYTE(psDiG2^.percenVal);  		   //发送DTD2比例阀值
	senddata[4] :=  WORD_TO_BYTE(SHR(psDiG2^.percenVal,8));    //0-65535  对应0-100  
	senddata[5] :=  WORD_TO_BYTE(psDiG3^.percenVal);  		   //发送DTD3比例阀值
	senddata[6] :=  WORD_TO_BYTE(SHR(psDiG3^.percenVal,8));    //0-65535  对应0-100  
	senddata[7] :=  WORD_TO_BYTE(psDiG4^.percenVal);  		   //发送DTD4比例阀值
	senddata[8] :=  WORD_TO_BYTE(SHR(psDiG4^.percenVal,8));    //0-65535  对应0-100  
	//发送至C0
	CAN_Send_Data_SWMC(1, 16#410,senddata);   //发送ID 0x410到C1
	
	2:
	 //C1-0x411
	senddata[1] :=  WORD_TO_BYTE(psDiG5^.percenVal);  		   //发送DTD5比例阀值
	senddata[2] :=  WORD_TO_BYTE(SHR(psDiG5^.percenVal,8));    //0-65535  对应0-100  
	
	senddata[3].0:=  psDiG1^.D00Q1.cmd.E_Open;               
	senddata[3].1:=  psDiG1^.D00Q2.cmd.R_Open;			//send D00Q1&D00Q2
	senddata[3].2:=  psDiG1^.D28L1.cmd.E_Open;               
	senddata[3].3:=  psDiG1^.D28L2.cmd.R_Open;			//send D28L1&D28L2
	
	senddata[4].0:=  psDiG1^.D29L.cmd.E_Open;               
	senddata[4].1:=  psDiG1^.D30L.cmd.R_Open;			//send D29L&D30L
	senddata[4].2:=  psDiG1^.D00L1.cmd.E_Open;               
	senddata[4].3:=  psDiG1^.D00L2.cmd.R_Open;			//send D00L1&00L2
	
	senddata[5].0:=  psDiG1^.D01L.cmd.E_Open;               
	senddata[5].1:=  psDiG1^.D01L.cmd.R_Open;           //send D01L
	senddata[5].2:=  psDiG1^.D28Q.cmd.E_Open;               
	senddata[5].3:=  psDiG1^.D29Q.cmd.R_Open;           //send D28Q&29Q
	
	senddata[6].0:=  psDiG1^.D30Q.cmd.E_Open;               
	senddata[6].1:=  psDiG1^.D30Q.cmd.R_Open;           //send D30Q
	//发送至C0
	CAN_Send_Data_SWMC(1, 16#411,senddata);				//发送ID 0x411到C1
	
	3:
	 //C1.1 IO-0x412
	senddata[1].0:=  psDiG2^.D02L.cmd.E_Open;               
	senddata[1].1:=  psDiG2^.D03L.cmd.R_Open;           //send D02L&D03L||D04L
	
	senddata[2].0:=  psDiG3^.D01Q1.cmd.E_Open;               
	senddata[2].1:=  psDiG3^.D01Q2.cmd.R_Open; 	        //send D01Q1&D01Q2||02~04QX

	senddata[3].0:=  psDiG4^.D05Q1.cmd.E_Open;               
	senddata[3].1:=  psDiG4^.D05Q2.cmd.R_Open;			//send D05Q1&05Q2||06~08QX
		
	senddata[4].0:=  psDiG5^.D09Q1.cmd.E_Open;               
	senddata[4].1:=  psDiG5^.D09Q2.cmd.R_Open;			//send D09Q1&09Q2||10~12QX
	//发送至C0
	CAN_Send_Data_SWMC(1, 16#412,senddata);				//发送ID 0x412到C1.1
	
	4:
	 //C1.2 IO-0x413
	senddata[1].0:=  psDiG2^.D05L.cmd.E_Open;               
	senddata[1].1:=  psDiG2^.D05L.cmd.R_Open;           //send D05L
	
	senddata[2].0:=  psDiG2^.D06L.cmd.E_Open;               
	senddata[2].1:=  psDiG2^.D07L.cmd.R_Open; 	        //send D06L&D07L||D08L

	senddata[3].0:=  psDiG2^.D09L.cmd.E_Open;               
	senddata[3].1:=  psDiG2^.D09L.cmd.R_Open;			//send D09L
		
	senddata[4].0:=  psDiG2^.D10L.cmd.E_Open;               
	senddata[4].1:=  psDiG2^.D11L.cmd.R_Open;			//send D010L&11L||D12L
	//发送至C0
	CAN_Send_Data_SWMC(1, 16#413,senddata);				//发送ID 0x413到C1.2

END_CASE

END_FUNCTION

// Device/Application/can/swmc_C02_Rx
FUNCTION swmc_C02_Rx : BOOL
VAR_INPUT
	CNT				: UINT;
	psYyz			: POINTER TO YyStation;
	
	psDiG7			: POINTER TO RatioValveD7;
END_VAR
VAR
	frame	 	    : Can_baseframe;
	COB_ID			: UINT;
	I				: UINT;
	pos				: WORD;
END_VAR

IF gCan.C2RxMsg.RxCounter <>  gCan.C2RxCounter THEN    //接收到新的数据

	FOR  I := 1 TO  gCan.C2RxMsg.NoOfRxMessages DO
		COB_ID :=	frame.id;    //获取ID
		CASE COB_ID OF     //根据ID解析协议
		
		
			//C1-0x320
			16#320:           //接收C2送来的数据
				pos := BYTE_TO_WORD(frame.data[1]) OR SHL(BYTE_TO_WORD(frame.data[2]),8);  	
				psDiG7^.D18L.status.posVal.Current:= pos*0.1;	//驱动插销油缸D18L-位移传感器	
				pos := BYTE_TO_WORD(frame.data[3]) OR SHL(BYTE_TO_WORD(frame.data[4]),8);  	
				psDig7^.D19L.status.posVal.Current:= pos*0.1;	//驱动插销油缸D19L-位移传感器	
				pos := BYTE_TO_WORD(frame.data[5]) OR SHL(BYTE_TO_WORD(frame.data[6]),8);  	
				psDig7^.D20L.status.posVal.Current:= pos*0.1;	//驱动插销油缸D20L-位移传感器		
				pos := BYTE_TO_WORD(frame.data[7]) OR SHL(BYTE_TO_WORD(frame.data[8]),8);  	
				psDig7^.D21L.status.posVal.Current:= pos*0.1;	//驱动插销油缸D21L-位移传感器		
			//C1-0x321
			16#321:           //接收C2送来的数据
				pos := BYTE_TO_WORD(frame.data[1]) OR SHL(BYTE_TO_WORD(frame.data[2]),8);  	
				psDig7^.D22L.status.posVal.Current:= pos*0.1;	//驱动插销油缸D22L-位移传感器	
				pos := BYTE_TO_WORD(frame.data[3]) OR SHL(BYTE_TO_WORD(frame.data[4]),8);  	
				psDig7^.D23L.status.posVal.Current:= pos*0.1;	//驱动插销油缸D23L-位移传感器	
				pos := BYTE_TO_WORD(frame.data[5]) OR SHL(BYTE_TO_WORD(frame.data[6]),8);  	
				psDig7^.D24L.status.posVal.Current:= pos*0.1;	//驱动插销油缸D24L-位移传感器	
				pos := BYTE_TO_WORD(frame.data[7]) OR SHL(BYTE_TO_WORD(frame.data[8]),8);  	
				psDig7^.D25L.status.posVal.Current:= pos*0.1;	//驱动插销油缸D25L-位移传感器
			//C1-0x322
			16#322:           //接收C2送来的数据
				pos := BYTE_TO_WORD(frame.data[1]) OR SHL(BYTE_TO_WORD(frame.data[2]),8);  	
				psDig7^.D26L.status.posVal.Current:= pos*0.1;	//驱动插销油缸D26L-位移传感器	
				pos := BYTE_TO_WORD(frame.data[3]) OR SHL(BYTE_TO_WORD(frame.data[4]),8);  	
				psDig7^.D17Q.status.posVal.Current:= pos*0.1;	//驱动插销油缸D17Q-位移传感器	
				pos := BYTE_TO_WORD(frame.data[5]) OR SHL(BYTE_TO_WORD(frame.data[6]),8);  	
				psDig7^.D18Q.status.posVal.Current:= pos*0.1;	//驱动插销油缸D18Q-位移传感器	
				pos := BYTE_TO_WORD(frame.data[7]) OR SHL(BYTE_TO_WORD(frame.data[8]),8);  	
				psDig7^.D19Q.status.posVal.Current:= pos*0.1;	//驱动插销油缸D19Q-位移传感器
			16#323:           //接收C2送来的数据
				pos := BYTE_TO_WORD(frame.data[1]) OR SHL(BYTE_TO_WORD(frame.data[2]),8);  	
				psDig7^.D20Q.status.posVal.Current:= pos*0.1;	//驱动插销油缸D20Q-位移传感器	
				pos := BYTE_TO_WORD(frame.data[3]) OR SHL(BYTE_TO_WORD(frame.data[4]),8);  	
				psDig7^.D21Q.status.posVal.Current:= pos*0.1;	//驱动插销油缸D21Q-位移传感器	
				pos := BYTE_TO_WORD(frame.data[5]) OR SHL(BYTE_TO_WORD(frame.data[6]),8);  	
				psDig7^.D22Q.status.posVal.Current:= pos*0.1;	//驱动插销油缸D22Q-位移传感器	
				pos := BYTE_TO_WORD(frame.data[7]) OR SHL(BYTE_TO_WORD(frame.data[8]),8);  	
				psDig7^.D23Q.status.posVal.Current:= pos*0.1;	//驱动插销油缸D23Q-位移传感器
		
			16#324:           //接收C2送来的数据
				pos := BYTE_TO_WORD(frame.data[1]) OR SHL(BYTE_TO_WORD(frame.data[2]),8);  	
				psDig7^.D24Q.status.posVal.Current:= pos*0.1;	//驱动插销油缸D24Q-位移传感器	
				pos := BYTE_TO_WORD(frame.data[3]) OR SHL(BYTE_TO_WORD(frame.data[4]),8);  	
				psDig7^.D25Q.status.posVal.Current:= pos*0.1;	//驱动插销油缸D25Q-位移传感器	
				pos := BYTE_TO_WORD(frame.data[5]) OR SHL(BYTE_TO_WORD(frame.data[6]),8);  	
				psDig7^.D26Q.status.posVal.Current:= pos*0.1;	//驱动插销油缸D26Q-位移传感器	
				pos := BYTE_TO_WORD(frame.data[7]) OR SHL(BYTE_TO_WORD(frame.data[8]),8);  	
				psDig7^.D17L1.status.posVal.Current:= pos*0.1;	//驱动插销油缸D17L1-位移传感器
			
			16#325:           //接收C2送来的数据
				pos := BYTE_TO_WORD(frame.data[1]) OR SHL(BYTE_TO_WORD(frame.data[2]),8);  	
				psDig7^.D17L2.status.posVal.Current:= pos*0.1;	//驱动插销油缸D17L2-位移传感器	
				pos := BYTE_TO_WORD(frame.data[3]) OR SHL(BYTE_TO_WORD(frame.data[4]),8);  	
				psDig7^.D27L1.status.posVal.Current:= pos*0.1;	//驱动插销油缸D27L1-位移传感器	
				pos := BYTE_TO_WORD(frame.data[5]) OR SHL(BYTE_TO_WORD(frame.data[6]),8);  	
				psDig7^.D27L2.status.posVal.Current:= pos*0.1;	//驱动插销油缸D27L2-位移传感器	
			

		END_CASE
	END_FOR


	gCan.C2RxCounter := gCan.C2RxMsg.RxCounter ;
END_IF

END_FUNCTION

// Device/Application/can/swmc_C02_Tx
FUNCTION swmc_C02_Tx : BOOL
VAR_INPUT
	CNT				: UINT;
	psDiG6			: POINTER TO RatioValveD6;
	psDiG7			: POINTER TO RatioValveD7;
END_VAR
VAR
	senddata	: ARRAY[1..8] OF BYTE;
	Send_cnt	: UINT;
END_VAR

//速度控制--待定
Send_cnt :=  CNT MOD 3;

CASE Send_cnt OF
	
	1:
 	//C2-0x420
	senddata[1] :=  WORD_TO_BYTE(psDiG6^.percenVal);  		   //发送DTD6比例阀值
	senddata[2] :=  WORD_TO_BYTE(SHR(psDiG6^.percenVal,8));    //0-65535  对应0-100  

	senddata[3] :=  WORD_TO_BYTE(psDiG7^.percenVal);  		   //发送DTD7比例阀值
	senddata[4] :=  WORD_TO_BYTE(SHR(psDiG7^.percenVal,8));    //0-65535  对应0-100  
	
	senddata[5].0:=  psDiG6^.D13Q.cmd.E_Open;
	senddata[5].1:=  psDiG6^.D14Q.cmd.R_Open;			//send D13Q&14Q
	senddata[5].2:=  psDiG6^.D15Q.cmd.E_Open;
	senddata[5].3:=  psDiG6^.D15Q.cmd.R_Open;			//send D15Q
	
	senddata[6].0:=  psDiG6^.D13L.cmd.E_Open;
	senddata[6].1:=  psDiG6^.D14L.cmd.R_Open;			//send D13L&14L
	senddata[6].2:=  psDiG6^.D15L.cmd.E_Open;
	senddata[6].3:=  psDiG6^.D15L.cmd.R_Open;			//send D15L
	
	senddata[7].0:=  psDiG6^.D16L1.cmd.E_Open;
	senddata[7].1:=  psDiG6^.D16L2.cmd.R_Open;			//send D16L1&16L2
	senddata[7].2:=  psDiG7^.D18L.cmd.E_Open;
	senddata[7].3:=  psDiG7^.D19L.cmd.R_Open;			//send D18L&19L||L20~21L
	
	senddata[8].0:=  psDiG7^.D22L.cmd.E_Open;
	senddata[8].1:=  psDiG7^.D22L.cmd.R_Open;			//send D22L1&22L2
	senddata[8].2:=  psDiG7^.D23L.cmd.E_Open;
	senddata[8].3:=  psDiG7^.D24L.cmd.R_Open;			//send D23L&24L||25L~26L
	
	
	//发送至C2
	CAN_Send_Data_SWMC(2, 16#420,senddata);				//发送ID 0x420到C2
	
	2:
 	//C2-0x421
		
	senddata[1].0:=  psDiG7^.D18Q.cmd.E_Open;
	senddata[1].1:=  psDiG7^.D19Q.cmd.R_Open;			//send D18Q&19Q||20Q~21Q
	
	senddata[2].0:=  psDiG7^.D22Q.cmd.E_Open;
	senddata[2].1:=  psDiG7^.D23Q.cmd.R_Open;			//send D22Q&23Q||24Q~26Q
	
	senddata[3].0:=  psDiG7^.D17L1.cmd.E_Open;
	senddata[3].1:=  psDiG7^.D17L2.cmd.R_Open;			//send D17L1&17L2
	
	senddata[4].0:=  psDiG7^.D27L1.cmd.E_Open;
	senddata[4].1:=  psDiG7^.D27L2.cmd.R_Open;			//send D27L1&27L2
	
	//发送至C2.1-IO
	CAN_Send_Data_SWMC(2, 16#421,senddata);				//发送ID 0x420到C2.1-IO
	
	
END_CASE

END_FUNCTION

// Device/Application/can/swmc_C09_Rx
FUNCTION swmc_C09_Rx : BOOL
VAR_INPUT
	CNT				: UINT;
	psYyz			: POINTER TO YyStation;
	psDiG1			: POINTER TO RatioValveD1;
	psDiG2			: POINTER TO RatioValveD2;
END_VAR
VAR
	frame	 	    : Can_baseframe;
	COB_ID			: UINT;
	I				: UINT;
	pos				: WORD;
END_VAR

IF gCan.C9RxMsg.RxCounter <>  gCan.C9RxCounter THEN    //接收到新的数据

	FOR  I := 1 TO  gCan.C9RxMsg.NoOfRxMessages DO
		COB_ID :=	frame.id;    //获取ID
		CASE COB_ID OF     //根据ID解析协议
		
		//比例阀DTD1
			//C9-0x390
			16#390:           //接收C9送来的数据
				pos := BYTE_TO_WORD(frame.data[1]) OR SHL(BYTE_TO_WORD(frame.data[2]),8);  	
				psDiG1^.D28L1.status.posVal.Current:= pos*0.1;	//驱动插销油缸D28L1-位移传感器	
				pos := BYTE_TO_WORD(frame.data[3]) OR SHL(BYTE_TO_WORD(frame.data[4]),8);  	
				psDig1^.D28L2.status.posVal.Current:= pos*0.1;	//驱动插销油缸D28L2-位移传感器	
				pos := BYTE_TO_WORD(frame.data[5]) OR SHL(BYTE_TO_WORD(frame.data[6]),8);  	
				psDig1^.D29L.status.posVal.Current:= pos*0.1;	//驱动插销油缸D29L-位移传感器		
				pos := BYTE_TO_WORD(frame.data[7]) OR SHL(BYTE_TO_WORD(frame.data[8]),8);  	
				psDig1^.D30L.status.posVal.Current:= pos*0.1;	//驱动插销油缸D30L-位移传感器		
			
			16#391:           //接收C9送来的数据
				pos := BYTE_TO_WORD(frame.data[1]) OR SHL(BYTE_TO_WORD(frame.data[2]),8);  	
				psDiG1^.D01L.status.posVal.Current:= pos*0.1;	//驱动插销油缸D01L-位移传感器	
				pos := BYTE_TO_WORD(frame.data[3]) OR SHL(BYTE_TO_WORD(frame.data[4]),8);  	
				psDig1^.D28Q.status.posVal.Current:= pos*0.1;	//驱动插销油缸D28Q-位移传感器	
				pos := BYTE_TO_WORD(frame.data[5]) OR SHL(BYTE_TO_WORD(frame.data[6]),8);  	
				psDig1^.D29Q.status.posVal.Current:= pos*0.1;	//驱动插销油缸D29Q-位移传感器		
				pos := BYTE_TO_WORD(frame.data[7]) OR SHL(BYTE_TO_WORD(frame.data[8]),8);  	
				psDig1^.D30Q.status.posVal.Current:= pos*0.1;	//驱动插销油缸D30Q-位移传感器		
				
			16#392:           //接收C9送来的数据
				pos := BYTE_TO_WORD(frame.data[1]) OR SHL(BYTE_TO_WORD(frame.data[2]),8);  	
				psDiG1^.D00L1.status.posVal.Current:= pos*0.1;	//驱动插销油缸D00L1-位移传感器	
				pos := BYTE_TO_WORD(frame.data[3]) OR SHL(BYTE_TO_WORD(frame.data[4]),8);  	
				psDig2^.D02L.status.posVal.Current:= pos*0.1;	//驱动插销油缸D02L-位移传感器	
				pos := BYTE_TO_WORD(frame.data[5]) OR SHL(BYTE_TO_WORD(frame.data[6]),8);  	
				psDig2^.D03L.status.posVal.Current:= pos*0.1;	//驱动插销油缸D03L-位移传感器		
				pos := BYTE_TO_WORD(frame.data[7]) OR SHL(BYTE_TO_WORD(frame.data[8]),8);  	
				psDig2^.D04L.status.posVal.Current:= pos*0.1;	//驱动插销油缸D04L-位移传感器		
				
			16#393:           //接收C9送来的数据
				pos := BYTE_TO_WORD(frame.data[1]) OR SHL(BYTE_TO_WORD(frame.data[2]),8);  	
				psDiG2^.D05L.status.posVal.Current:= pos*0.1;	//驱动插销油缸D05L-位移传感器	
				pos := BYTE_TO_WORD(frame.data[3]) OR SHL(BYTE_TO_WORD(frame.data[4]),8);  	
				psDig2^.D06L.status.posVal.Current:= pos*0.1;	//驱动插销油缸D06L-位移传感器	
				pos := BYTE_TO_WORD(frame.data[5]) OR SHL(BYTE_TO_WORD(frame.data[6]),8);  	
				psDig2^.D07L.status.posVal.Current:= pos*0.1;	//驱动插销油缸D07L-位移传感器		
				pos := BYTE_TO_WORD(frame.data[7]) OR SHL(BYTE_TO_WORD(frame.data[8]),8);  	
				psDig2^.D08L.status.posVal.Current:= pos*0.1;	//驱动插销油缸D08L-位移传感器		

			16#394:           //接收C9送来的数据
				pos := BYTE_TO_WORD(frame.data[1]) OR SHL(BYTE_TO_WORD(frame.data[2]),8);  	
				psDiG2^.D09L.status.posVal.Current:= pos*0.1;	//驱动插销油缸D09L-位移传感器	
				pos := BYTE_TO_WORD(frame.data[3]) OR SHL(BYTE_TO_WORD(frame.data[4]),8);  	
				psDig2^.D10L.status.posVal.Current:= pos*0.1;	//驱动插销油缸D10L-位移传感器	
				pos := BYTE_TO_WORD(frame.data[5]) OR SHL(BYTE_TO_WORD(frame.data[6]),8);  	
				psDig2^.D11L.status.posVal.Current:= pos*0.1;	//驱动插销油缸D11L-位移传感器		
				pos := BYTE_TO_WORD(frame.data[7]) OR SHL(BYTE_TO_WORD(frame.data[8]),8);  	
				psDig2^.D12L.status.posVal.Current:= pos*0.1;	//驱动插销油缸D12L-位移传感器		
				
			16#395:           //接收C9送来的数据
				pos := BYTE_TO_WORD(frame.data[1]) OR SHL(BYTE_TO_WORD(frame.data[2]),8);  	
				psDiG1^.D00L2.status.posVal.Current:= pos*0.1;	//驱动插销油缸D00L2-位移传感器	
				pos := BYTE_TO_WORD(frame.data[3]) OR SHL(BYTE_TO_WORD(frame.data[4]),8);  	
				psDig1^.D00Q1.status.posVal.Current:= pos*0.1;	//驱动插销油缸D00Q1-位移传感器	
				pos := BYTE_TO_WORD(frame.data[5]) OR SHL(BYTE_TO_WORD(frame.data[6]),8);  	
				psDig1^.D00Q2.status.posVal.Current:= pos*0.1;	//驱动插销油缸D00Q2-位移传感器		
		END_CASE
	END_FOR


	gCan.C0RxCounter := gCan.C0RxMsg.RxCounter ;
END_IF

END_FUNCTION

// Device/Application/can/swmc_C10_Rx
FUNCTION swmc_C10_Rx : BOOL
VAR_INPUT
	CNT				: UINT;
	psYyz			: POINTER TO YyStation;
	psDiG6			: POINTER TO RatioValveD6;

END_VAR
VAR
	frame	 	    : Can_baseframe;
	COB_ID			: UINT;
	I				: UINT;
	pos				: WORD;
END_VAR

IF gCan.C10RxMsg.RxCounter <>  gCan.C10RxCounter THEN    //接收到新的数据

	FOR  I := 1 TO  gCan.C10RxMsg.NoOfRxMessages DO
		COB_ID :=	frame.id;    //获取ID
		CASE COB_ID OF     //根据ID解析协议
			//C10-0x3A0
			16#3A0:           //接收C10送来的数据
				pos := BYTE_TO_WORD(frame.data[1]) OR SHL(BYTE_TO_WORD(frame.data[2]),8);  	
				psDiG6^.D13Q.status.posVal.Current:= pos*0.1;	//驱动插销油缸D13Q-位移传感器	
				pos := BYTE_TO_WORD(frame.data[3]) OR SHL(BYTE_TO_WORD(frame.data[4]),8);  	
				psDig6^.D14Q.status.posVal.Current:= pos*0.1;	//驱动插销油缸D14Q-位移传感器	
				pos := BYTE_TO_WORD(frame.data[5]) OR SHL(BYTE_TO_WORD(frame.data[6]),8);  	
				psDig6^.D15Q.status.posVal.Current:= pos*0.1;	//驱动插销油缸D15Q-位移传感器		
				pos := BYTE_TO_WORD(frame.data[7]) OR SHL(BYTE_TO_WORD(frame.data[8]),8);  	
				psDig6^.D16L1.status.posVal.Current:= pos*0.1;	//驱动插销油缸D16L1-位移传感器		
			//C10-0x3A1
			16#3A1:           //接收C10送来的数据
				pos := BYTE_TO_WORD(frame.data[1]) OR SHL(BYTE_TO_WORD(frame.data[2]),8);  	
				psDiG6^.D13L.status.posVal.Current:= pos*0.1;	//驱动插销油缸D13L-位移传感器	
				pos := BYTE_TO_WORD(frame.data[3]) OR SHL(BYTE_TO_WORD(frame.data[4]),8);  	
				psDig6^.D14L.status.posVal.Current:= pos*0.1;	//驱动插销油缸D14L-位移传感器	
				pos := BYTE_TO_WORD(frame.data[5]) OR SHL(BYTE_TO_WORD(frame.data[6]),8);  	
				psDig6^.D15L.status.posVal.Current:= pos*0.1;	//驱动插销油缸D15L-位移传感器		
				pos := BYTE_TO_WORD(frame.data[7]) OR SHL(BYTE_TO_WORD(frame.data[8]),8);  	
				psDig6^.D16L2.status.posVal.Current:= pos*0.1;	//驱动插销油缸D16L2-位移传感器		
			
		END_CASE
	END_FOR


	gCan.C10RxCounter := gCan.C10RxMsg.RxCounter ;
END_IF

END_FUNCTION

// Device/Application/display/YY_Station_Display
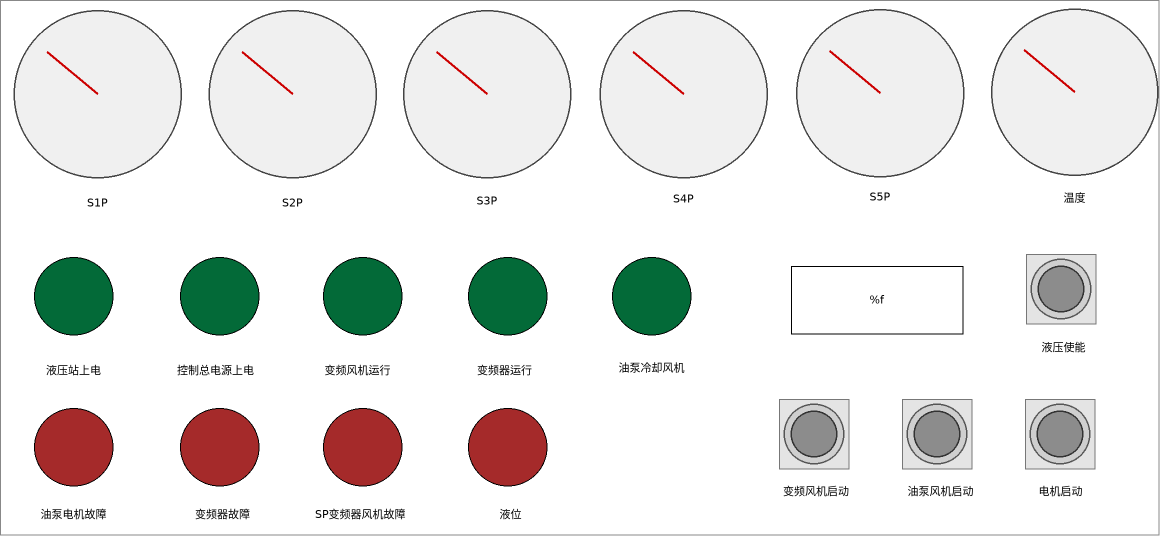
VISUALIZATION YY_Station_Display  // 1160x536
    Meter360 (10,10 175x168), value: gUI.rPressureVal1, style: Meter-Meter360-Gray, scale format: %.1f, scale 0..100
        p518627256: bar
    Meter360 (206,10 173x168), value: gUI.rPressureVal2, style: Meter-Meter360-Gray, scale format: %.1f, scale 0..100
        p518627256: bar
    Meter360 (402,10 170x168), value: gUI.rPressureVal3, style: Meter-Meter360-Gray, scale format: %.1f, scale 0..100
        p518627256: bar
    Meter360 (598,10 171x168), value: gUI.rPressureVal4, style: Meter-Meter360-Gray, scale format: %.1f, scale 0..100
        p518627256: bar
    Meter360 (796,9 168x168), value: gUI.rPressureVal5, style: Meter-Meter360-Gray, scale format: %.1f, scale 0..200
        p518627256: bar
    Label (10,188 175x30), "S1P"
    Label (206,188 173x30), "S2P"
    Label (402,186 170x30), "S3P"
    Label (598,184 171x30), "S4P"
    Label (796,182 168x30), "S5P"
    Ellipse (34,257 79x78), colour toggle: gUI.bYysPower
    Ellipse (180,257 79x78), colour toggle: gUI.bCtrlPower
    Ellipse (323,257 79x78), colour toggle: gUI.bFreqConverterFan
    Ellipse (468,257 79x78), colour toggle: gUI.bFreqConverter
    Label (-4,351 155x39), "液压站上电"
    Label (138,351 155x39), "控制总电源上电"
    Label (280,351 155x39), "变频风机运行"
    Label (465,351 79x39), "变频器运行"
    Ellipse (34,408 79x78), colour toggle: gUI.bOilPumpM_Fault
    Ellipse (180,408 79x78), colour toggle: gUI.bFreqConverter_Fault
    Label (34,495 79x39), "油泵电机故障"
    Label (612,351 79x34), "油泵冷却风机"
    Label (145,495 155x39), "变频器故障"
    Ellipse (323,408 79x78), colour toggle: gUI.bFreqConverterFan_Fault
    Label (283,495 155x39), "SP变频器风机故障"
    Ellipse (468,408 79x78), colour toggle: gUI.bFluidLevel
    Label (471,495 79x39), "液位"
    Meter360 (991,8 167x168), value: gUI.rPressureVal5, style: Meter-Meter360-Gray, scale format: %.1f, scale 0..200
        p518627256: bar
    Label (991,183 167x30), "温度"
    PushSwitchLed (779,399 70x70), variable: gUI.cmdInverterFan, behaviour: TOGGLE, style: Switch-PushSwitchLed-Gray
    PushSwitchLed (902,399 70x70), variable: gUI.cmdOilPumpFan, behaviour: TOGGLE, style: Switch-PushSwitchLed-Gray
    Label (768,472 96x39), "变频风机启动"
    Label (863,472 155x39), "油泵风机启动"
    PushSwitchLed (1025,399 70x70), variable: gUI.cmdOilPumpM, behaviour: TOGGLE, style: Switch-PushSwitchLed-Gray
    Label (983,472 155x39), "电机启动"
    Rectangle (791,266 172x68), "%f", text variable: gUI.cmdOilPrePercent
        OnMouseDown: write the text variable via Default, min 0, max 100
    Label (986,328 155x39), "液压使能"
    PushSwitchLed (1026,254 70x70), variable: gUI.cmdOilPre_EN, behaviour: TOGGLE, style: Switch-PushSwitchLed-Gray
    Ellipse (612,257 79x78), colour toggle: gUI.bFreqConverter
END_VISUALIZATION

// Device/Application/display/Orig/Module/OilBlock_PrimButton
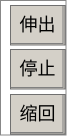
VISUALIZATION OilBlock_PrimButton  // 67x136
VAR_IN_OUT
	extendButton		: BOOL;
	retractButton		: BOOL;
	stopButton			: BOOL;
	
END_VAR
    Button (10,94 55x40), "缩回"
        toggle retractButton
    Button (10,49 55x40), "停止"
        toggle stopButton
    Button (10,5 55x40), "伸出"
        toggle extendButton
END_VISUALIZATION

// Device/Application/display/Orig/Module/OilBlock_PrimInfo
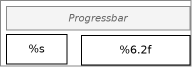
VISUALIZATION OilBlock_PrimInfo  // 192x67
VAR_IN_OUT
	nameStr		:STRING;
	posVal		:REAL;
	percentBar	:REAL;
END_VAR
    RoundedRectangle (6,34 61x30), "%s", text variable: nameStr
    RoundedRectangle (81,35 109x30), "%6.2f", text variable: posVal
    Progressbar (6,6 184x24), variable: percentBar
END_VISUALIZATION

// Device/Application/display/Orig/Floor_Rail1
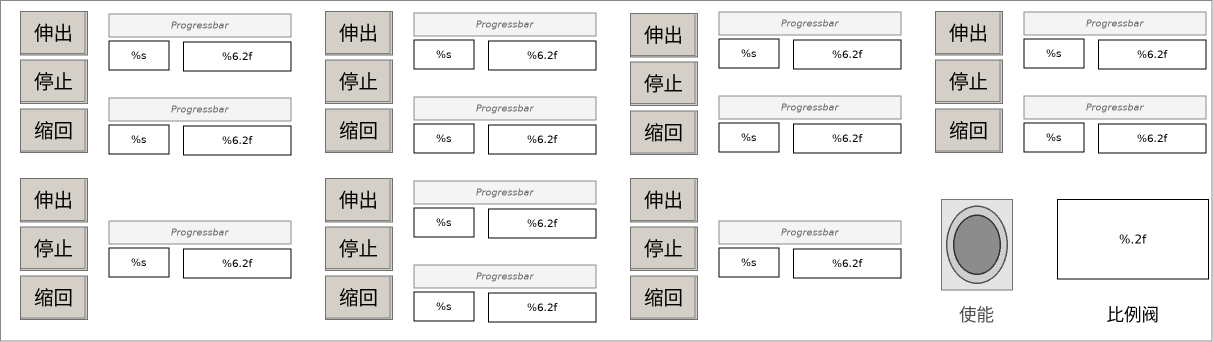
VISUALIZATION Floor_Rail1  // 1213x342
    Group (8,6 285x151)
        Frame (0,0 82x149)
            shows OilBlock_PrimButton(extendButton := gUI.DiG1.S1.bExtend, retractButton := gUI.DiG1.S1.bRetract, stopButton := gUI.DiG1.S1.bStop)
        Group (95,2 190x149)
            Frame (0,0 190x65)
                shows OilBlock_PrimInfo(nameStr := gUI.DiG1.D00Q1.strName, posVal := gUI.DiG1.D00Q1.rPosition, percentBar := gUI.DiG1.D00Q1.rPercent)
            Frame (0,84 190x65)
                shows OilBlock_PrimInfo(nameStr := gUI.DiG1.D00Q2.strName, posVal := gUI.DiG1.D00Q2.rPosition, percentBar := gUI.DiG1.D00Q2.rPercent)
    Group (313,6 285x150)
        Group (95,1 190x149)
            Frame (0,0 190x65)
                shows OilBlock_PrimInfo(nameStr := gUI.DiG1.D28L1.strName, posVal := gUI.DiG1.D28L1.rPosition, percentBar := gUI.DiG1.D28L1.rPercent)
            Frame (0,84 190x65)
                shows OilBlock_PrimInfo(nameStr := gUI.DiG1.D28L2.strName, posVal := gUI.DiG1.D28L2.rPosition, percentBar := gUI.DiG1.D28L2.rPercent)
        Frame (0,0 82x149)
            shows OilBlock_PrimButton(extendButton := gUI.DiG1.S2.bExtend, retractButton := gUI.DiG1.S2.bRetract, stopButton := gUI.DiG1.S2.bStop)
    Group (618,6 285x151)
        Group (95,0 190x149)
            Frame (0,0 190x65)
                shows OilBlock_PrimInfo(nameStr := gUI.DiG1.D29L.strName, posVal := gUI.DiG1.D29L.rPosition, percentBar := gUI.DiG1.D29L.rPercent)
            Frame (0,84 190x65)
                shows OilBlock_PrimInfo(nameStr := gUI.DiG1.D30L.strName, posVal := gUI.DiG1.D30L.rPosition, percentBar := gUI.DiG1.D30L.rPercent)
        Frame (0,2 82x149)
            shows OilBlock_PrimButton(extendButton := gUI.DiG1.S3.bExtend, retractButton := gUI.DiG1.S3.bRetract, stopButton := gUI.DiG1.S3.bStop)
    Group (923,6 285x149)
        Group (95,0 190x149)
            Frame (0,0 190x65)
                shows OilBlock_PrimInfo(nameStr := gUI.DiG1.D00L1.strName, posVal := gUI.DiG1.D00L1.rPosition, percentBar := gUI.DiG1.D00L1.rPercent)
            Frame (0,84 190x65)
                shows OilBlock_PrimInfo(nameStr := gUI.DiG1.D00L2.strName, posVal := gUI.DiG1.D00L2.rPosition, percentBar := gUI.DiG1.D00L2.rPercent)
        Frame (0,0 82x149)
            shows OilBlock_PrimButton(extendButton := gUI.DiG1.S4.bExtend, retractButton := gUI.DiG1.S4.bRetract, stopButton := gUI.DiG1.S4.bStop)
    Frame (103,215 190x65)
        shows OilBlock_PrimInfo(nameStr := gUI.DiG1.D01L.strName, posVal := gUI.DiG1.D01L.rPosition, percentBar := gUI.DiG1.D01L.rPercent)
    Frame (8,173 82x149)
        shows OilBlock_PrimButton(extendButton := gUI.DiG1.S5.bExtend, retractButton := gUI.DiG1.S5.bRetract, stopButton := gUI.DiG1.S5.bStop)
    Group (313,173 285x151)
        Group (95,2 190x149)
            Frame (0,0 190x65)
                shows OilBlock_PrimInfo(nameStr := gUI.DiG1.D28Q.strName, posVal := gUI.DiG1.D28Q.rPosition, percentBar := gUI.DiG1.D28Q.rPercent)
            Frame (0,84 190x65)
                shows OilBlock_PrimInfo(nameStr := gUI.DiG1.D29Q.strName, posVal := gUI.DiG1.D29Q.rPosition, percentBar := gUI.DiG1.D29Q.rPercent)
        Frame (0,0 82x149)
            shows OilBlock_PrimButton(extendButton := gUI.DiG1.S6.bExtend, retractButton := gUI.DiG1.S6.bRetract, stopButton := gUI.DiG1.S6.bStop)
    Group (618,173 285x149)
        Frame (95,42 190x65)
            shows OilBlock_PrimInfo(nameStr := gUI.DiG1.D30Q.strName, posVal := gUI.DiG1.D30Q.rPosition, percentBar := gUI.DiG1.D30Q.rPercent)
        Frame (0,0 82x149)
            shows OilBlock_PrimButton(extendButton := gUI.DiG1.S7.bExtend, retractButton := gUI.DiG1.S7.bRetract, stopButton := gUI.DiG1.S7.bStop)
    Frame (926,191 285x149)
        shows ModuleDTD(enable := gUI.DiG1.bRVD1_enable, propPercent := gUI.DiG1.rRVD1Percent)
END_VISUALIZATION

// Device/Application/display/Orig/Module/ModuleX2
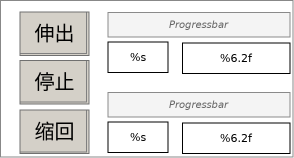
VISUALIZATION ModuleX2  // 294x158
VAR_IN_OUT
	extendButton		: BOOL;
	retractButton		: BOOL;
	stopButton			: BOOL;
	
	nameStr1			:STRING;
	posVal1				:REAL;
	percentBar1			:REAL;
	nameStr2			:STRING;
	posVal2				:REAL;
	percentBar2			:REAL;
END_VAR
    Frame (7,6 85x150)
        shows OilBlock_PrimButton(extendButton := extendButton, retractButton := retractButton, stopButton := stopButton)
    Frame (102,6 190x70)
        shows OilBlock_PrimInfo(nameStr := nameStr1, posVal := posVal1, percentBar := percentBar1)
    Frame (102,86 190x70)
        shows OilBlock_PrimInfo(nameStr := nameStr2, posVal := posVal2, percentBar := percentBar2)
END_VISUALIZATION

// Device/Application/display/Orig/Module/ModuleX1
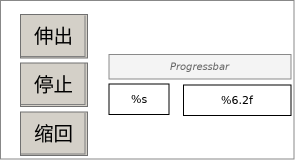
VISUALIZATION ModuleX1  // 295x160
VAR_IN_OUT
	extendButton		: BOOL;
	retractButton		: BOOL;
	stopButton			: BOOL;
	
	nameStr				:STRING;
	posVal				:REAL;
	percentBar			:REAL;
END_VAR
    Frame (8,9 82x149)
        shows OilBlock_PrimButton(extendButton := extendButton, retractButton := retractButton, stopButton := stopButton)
    Frame (103,48 190x70)
        shows OilBlock_PrimInfo(nameStr := nameStr, posVal := posVal, percentBar := percentBar)
END_VISUALIZATION

// Device/Application/display/Orig/Module/ModuleX3
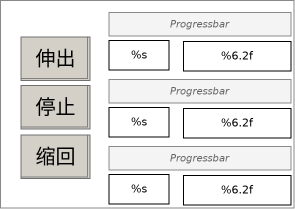
VISUALIZATION ModuleX3  // 295x209
VAR_IN_OUT
	extendButton		: BOOL;
	retractButton		: BOOL;
	stopButton			: BOOL;
	
	nameStr1			:STRING;
	posVal1				:REAL;
	percentBar1			:REAL;
	nameStr2			:STRING;
	posVal2				:REAL;
	percentBar2			:REAL;
	nameStr3			:STRING;
	posVal3				:REAL;
	percentBar3			:REAL;
END_VAR
    Frame (8,31 85x150)
        shows OilBlock_PrimButton(extendButton := extendButton, retractButton := retractButton, stopButton := stopButton)
    Frame (103,6 190x67)
        shows OilBlock_PrimInfo(nameStr := nameStr1, posVal := posVal1, percentBar := percentBar1)
    Frame (103,73 190x67)
        shows OilBlock_PrimInfo(nameStr := nameStr2, posVal := posVal2, percentBar := percentBar2)
    Frame (103,140 190x67)
        shows OilBlock_PrimInfo(nameStr := nameStr3, posVal := posVal3, percentBar := percentBar3)
END_VISUALIZATION

// Device/Application/display/Orig/Module/ModuleX8
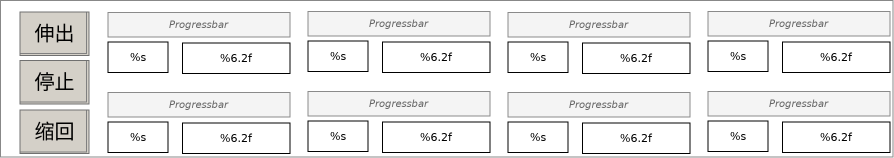
VISUALIZATION ModuleX8  // 894x158
VAR_IN_OUT
	extendButton		: BOOL;
	retractButton		: BOOL;
	stopButton			: BOOL;
	
	nameStr1			:STRING;
	posVal1				:REAL;
	percentBar1			:REAL;
	
	nameStr2			:STRING;
	posVal2				:REAL;
	percentBar2			:REAL;
	
	nameStr3			:STRING;
	posVal3				:REAL;
	percentBar3			:REAL;
	
	nameStr4			:STRING;
	posVal4				:REAL;
	percentBar4			:REAL;
	
	nameStr5			:STRING;
	posVal5				:REAL;
	percentBar5			:REAL;
	
	nameStr6			:STRING;
	posVal6				:REAL;
	percentBar6			:REAL;
	
	nameStr7			:STRING;
	posVal7				:REAL;
	percentBar7			:REAL;
	
	nameStr8			:STRING;
	posVal8				:REAL;
	percentBar8			:REAL;	
	
END_VAR
    Frame (7,6 85x150)
        shows OilBlock_PrimButton(extendButton := extendButton, retractButton := retractButton, stopButton := stopButton)
    Group (102,5 390x151)
        Group (0,1 190x150)
            Frame (0,0 190x70)
                shows OilBlock_PrimInfo(nameStr := nameStr1, posVal := posVal1, percentBar := percentBar1)
            Frame (0,80 190x70)
                shows OilBlock_PrimInfo(nameStr := nameStr2, posVal := posVal2, percentBar := percentBar2)
        Frame (200,0 190x70)
            shows OilBlock_PrimInfo(nameStr := nameStr3, posVal := posVal3, percentBar := percentBar3)
        Frame (200,80 190x70)
            shows OilBlock_PrimInfo(nameStr := nameStr4, posVal := posVal4, percentBar := percentBar4)
    Frame (502,6 190x70)
        shows OilBlock_PrimInfo(nameStr := nameStr5, posVal := posVal5, percentBar := percentBar5)
    Frame (502,86 190x70)
        shows OilBlock_PrimInfo(nameStr := nameStr6, posVal := posVal6, percentBar := percentBar6)
    Frame (702,5 190x70)
        shows OilBlock_PrimInfo(nameStr := nameStr7, posVal := posVal7, percentBar := percentBar7)
    Frame (702,85 190x70)
        shows OilBlock_PrimInfo(nameStr := nameStr8, posVal := posVal8, percentBar := percentBar8)
END_VISUALIZATION

// Device/Application/display/Orig/Module/ModuleX4
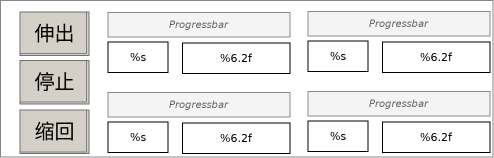
VISUALIZATION ModuleX4  // 494x158
VAR_IN_OUT
	extendButton		: BOOL;
	retractButton		: BOOL;
	stopButton			: BOOL;
	
	nameStr1			:STRING;
	posVal1				:REAL;
	percentBar1			:REAL;
	nameStr2			:STRING;
	posVal2				:REAL;
	percentBar2			:REAL;
	nameStr3			:STRING;
	posVal3				:REAL;
	percentBar3			:REAL;
	nameStr4			:STRING;
	posVal4				:REAL;
	percentBar4			:REAL;
	
	
END_VAR
    Frame (7,6 85x150)
        shows OilBlock_PrimButton(extendButton := extendButton, retractButton := retractButton, stopButton := stopButton)
    Group (102,6 190x150)
        Frame (0,0 190x70)
            shows OilBlock_PrimInfo(nameStr := nameStr1, posVal := posVal1, percentBar := percentBar1)
        Frame (0,80 190x70)
            shows OilBlock_PrimInfo(nameStr := nameStr2, posVal := posVal2, percentBar := percentBar2)
    Frame (302,5 190x70)
        shows OilBlock_PrimInfo(nameStr := nameStr3, posVal := posVal3, percentBar := percentBar3)
    Frame (302,85 190x70)
        shows OilBlock_PrimInfo(nameStr := nameStr4, posVal := posVal4, percentBar := percentBar4)
END_VISUALIZATION

// Device/Application/display/Orig/Module/ModuleX5
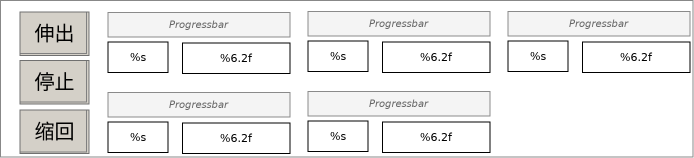
VISUALIZATION ModuleX5  // 694x158
VAR_IN_OUT
	extendButton		: BOOL;
	retractButton		: BOOL;
	stopButton			: BOOL;
	
	nameStr1			:STRING;
	posVal1				:REAL;
	percentBar1			:REAL;
	nameStr2			:STRING;
	posVal2				:REAL;
	percentBar2			:REAL;
	nameStr3			:STRING;
	posVal3				:REAL;
	percentBar3			:REAL;
	nameStr4			:STRING;
	posVal4				:REAL;
	percentBar4			:REAL;
	nameStr5			:STRING;
	posVal5				:REAL;
	percentBar5			:REAL;
	
	
END_VAR
    Frame (7,6 85x150)
        shows OilBlock_PrimButton(extendButton := extendButton, retractButton := retractButton, stopButton := stopButton)
    Group (102,6 190x150)
        Frame (0,0 190x70)
            shows OilBlock_PrimInfo(nameStr := nameStr1, posVal := posVal1, percentBar := percentBar1)
        Frame (0,80 190x70)
            shows OilBlock_PrimInfo(nameStr := nameStr2, posVal := posVal2, percentBar := percentBar2)
    Frame (302,5 190x70)
        shows OilBlock_PrimInfo(nameStr := nameStr3, posVal := posVal3, percentBar := percentBar3)
    Frame (302,85 190x70)
        shows OilBlock_PrimInfo(nameStr := nameStr4, posVal := posVal4, percentBar := percentBar4)
    Frame (502,5 190x70)
        shows OilBlock_PrimInfo(nameStr := nameStr5, posVal := posVal5, percentBar := percentBar5)
END_VISUALIZATION

// Device/Application/display/Orig/Floor_Rail2
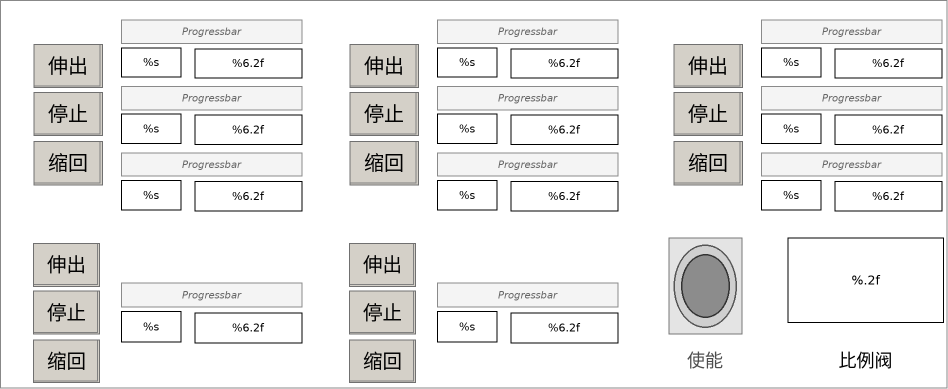
VISUALIZATION Floor_Rail2  // 948x389
    Frame (13,8 293x207)
        shows ModuleX3(extendButton := gUI.DiG2.S1.bExtend, retractButton := gUI.DiG2.S1.bRetract, stopButton := gUI.DiG2.S1.bStop, nameStr1 := gUI.DiG2.D02L.strName, posVal1 := gUI.DiG2.D02L.rPosition, percentBar1 := gUI.DiG2.D02L.rPercent, nameStr2 := gUI.DiG2.D03L.strName, posVal2 := gUI.DiG2.D03L.rPosition, percentBar2 := gUI.DiG2.D03L.rPercent, nameStr3 := gUI.DiG2.D04L.strName, posVal3 := gUI.DiG2.D04L.rPosition, percentBar3 := gUI.DiG2.D04L.rPercent)
    Frame (13,229 293x158)
        shows ModuleX1(extendButton := gUI.DiG2.S2.bExtend, retractButton := gUI.DiG2.S2.bRetract, stopButton := gUI.DiG2.S2.bStop, nameStr := gUI.DiG2.D05L.strName, posVal := gUI.DiG2.D05L.rPosition, percentBar := gUI.DiG2.D05L.rPercent)
    Frame (329,8 293x207)
        shows ModuleX3(extendButton := gUI.DiG2.S3.bExtend, retractButton := gUI.DiG2.S3.bRetract, stopButton := gUI.DiG2.S3.bStop, nameStr1 := gUI.DiG2.D06L.strName, posVal1 := gUI.DiG2.D06L.rPosition, percentBar1 := gUI.DiG2.D06L.rPercent, nameStr2 := gUI.DiG2.D07L.strName, posVal2 := gUI.DiG2.D07L.rPosition, percentBar2 := gUI.DiG2.D07L.rPercent, nameStr3 := gUI.DiG2.D08L.strName, posVal3 := gUI.DiG2.D08L.rPosition, percentBar3 := gUI.DiG2.D08L.rPercent)
    Frame (329,229 293x158)
        shows ModuleX1(extendButton := gUI.DiG2.S4.bExtend, retractButton := gUI.DiG2.S4.bRetract, stopButton := gUI.DiG2.S4.bStop, nameStr := gUI.DiG2.D09L.strName, posVal := gUI.DiG2.D09L.rPosition, percentBar := gUI.DiG2.D09L.rPercent)
    Frame (653,8 293x207)
        shows ModuleX3(extendButton := gUI.DiG2.S5.bExtend, retractButton := gUI.DiG2.S5.bRetract, stopButton := gUI.DiG2.S5.bStop, nameStr1 := gUI.DiG2.D10L.strName, posVal1 := gUI.DiG2.D10L.rPosition, percentBar1 := gUI.DiG2.D10L.rPercent, nameStr2 := gUI.DiG2.D11L.strName, posVal2 := gUI.DiG2.D11L.rPosition, percentBar2 := gUI.DiG2.D11L.rPercent, nameStr3 := gUI.DiG2.D12L.strName, posVal3 := gUI.DiG2.D12L.rPosition, percentBar3 := gUI.DiG2.D12L.rPercent)
    Frame (653,229 293x158)
        shows ModuleDTD(enable := gUI.DiG2.bRVD2_enable, propPercent := gUI.DiG2.rRVD2Percent)
END_VISUALIZATION

// Device/Application/display/Orig/Module/ModuleDTD
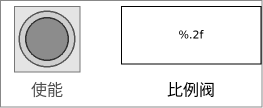
VISUALIZATION ModuleDTD  // 263x108
VAR_IN_OUT
	enable			:BOOL;
	propPercent		:REAL;
END_VAR
    Rectangle (121,6 140x58), "%.2f", text variable: propPercent
        OnMouseDown: write the text variable via Default, min 0, max 100
    Label (121,74 140x32), "比例阀"
    PushSwitchLed (13,6 68x66), variable: enable, behaviour: TOGGLE, style: Switch-PushSwitchLed-Gray
    Label (13,74 68x32), "使能"
END_VISUALIZATION

// Device/Application/display/Orig/Floor_Rail_345
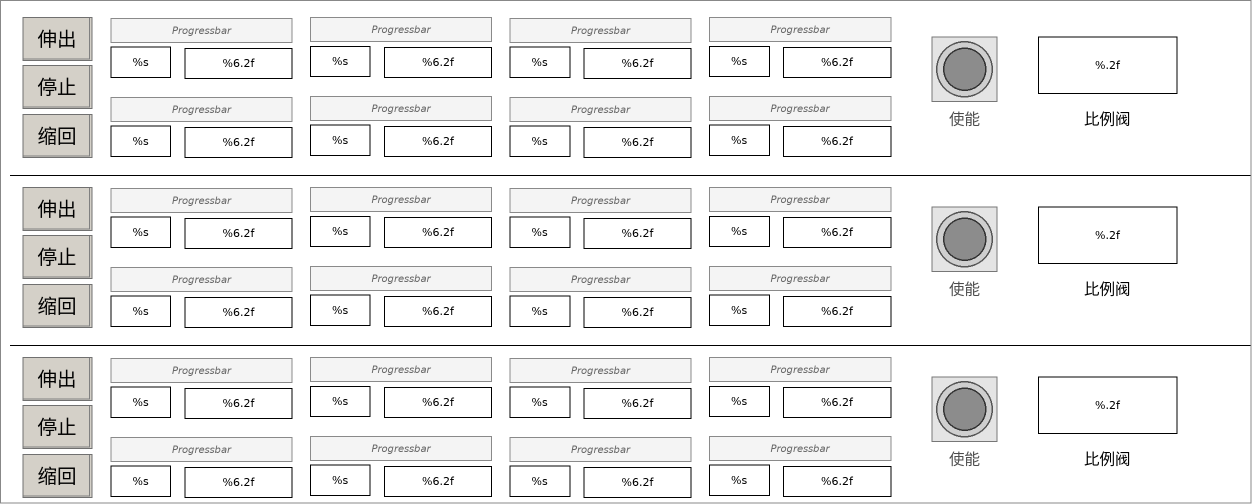
VISUALIZATION Floor_Rail_345  // 1252x504
    Frame (3,6 892x156)
        shows ModuleX8(extendButton := gUI.DiG3.S1.bExtend, retractButton := gUI.DiG3.S1.bRetract, stopButton := gUI.DiG3.S1.bStop, nameStr1 := gUI.DiG3.D01Q1.strName, posVal1 := gUI.DiG3.D01Q1.rPosition, percentBar1 := gUI.DiG3.D01Q1.rPercent, nameStr2 := gUI.DiG3.D01Q2.strName, posVal2 := gUI.DiG3.D01Q2.rPosition, percentBar2 := gUI.DiG3.D01Q2.rPercent, nameStr3 := gUI.DiG3.D02Q1.strName, posVal3 := gUI.DiG3.D02Q1.rPosition, percentBar3 := gUI.DiG3.D02Q1.rPercent, nameStr4 := gUI.DiG3.D02Q2.strName, posVal4 := gUI.DiG3.D02Q2.rPosition, percentBar4 := gUI.DiG3.D02Q2.rPercent, nameStr5 := gUI.DiG3.D03Q1.strName, posVal5 := gUI.DiG3.D03Q1.rPosition, percentBar5 := gUI.DiG3.D03Q1.rPercent, nameStr6 := gUI.DiG3.D03Q2.strName, posVal6 := gUI.DiG3.D03Q2.rPosition, percentBar6 := gUI.DiG3.D03Q2.rPercent, nameStr7 := gUI.DiG3.D04Q1.strName, posVal7 := gUI.DiG3.D04Q1.rPosition, percentBar7 := gUI.DiG3.D04Q1.rPercent, nameStr8 := gUI.DiG3.D04Q2.strName, posVal8 := gUI.DiG3.D04Q2.rPosition, percentBar8 := gUI.DiG3.D04Q2.rPercent)
    Frame (3,176 892x156)
        shows ModuleX8(extendButton := gUI.DiG4.S1.bExtend, retractButton := gUI.DiG4.S1.bRetract, stopButton := gUI.DiG4.S1.bStop, nameStr1 := gUI.DiG4.D05Q1.strName, posVal1 := gUI.DiG4.D05Q1.rPosition, percentBar1 := gUI.DiG4.D05Q1.rPercent, nameStr2 := gUI.DiG4.D05Q2.strName, posVal2 := gUI.DiG4.D05Q2.rPosition, percentBar2 := gUI.DiG4.D05Q2.rPercent, nameStr3 := gUI.DiG4.D06Q1.strName, posVal3 := gUI.DiG4.D06Q1.rPosition, percentBar3 := gUI.DiG4.D06Q1.rPercent, nameStr4 := gUI.DiG4.D06Q2.strName, posVal4 := gUI.DiG4.D06Q2.rPosition, percentBar4 := gUI.DiG4.D06Q2.rPercent, nameStr5 := gUI.DiG4.D07Q1.strName, posVal5 := gUI.DiG4.D07Q1.rPosition, percentBar5 := gUI.DiG4.D07Q1.rPercent, nameStr6 := gUI.DiG4.D07Q2.strName, posVal6 := gUI.DiG4.D07Q2.rPosition, percentBar6 := gUI.DiG4.D07Q2.rPercent, nameStr7 := gUI.DiG4.D08Q1.strName, posVal7 := gUI.DiG4.D08Q1.rPosition, percentBar7 := gUI.DiG4.D08Q1.rPercent, nameStr8 := gUI.DiG4.D08Q2.strName, posVal8 := gUI.DiG4.D08Q2.rPosition, percentBar8 := gUI.DiG4.D08Q2.rPercent)
    Frame (3,346 892x156)
        shows ModuleX8(extendButton := gUI.DiG5.S1.bExtend, retractButton := gUI.DiG5.S1.bStop, stopButton := gUI.DiG5.S1.bStop, nameStr1 := gUI.DiG5.D09Q1.strName, posVal1 := gUI.DiG5.D09Q1.rPosition, percentBar1 := gUI.DiG5.D09Q1.rPercent, nameStr2 := gUI.DiG5.D09Q2.strName, posVal2 := gUI.DiG5.D09Q2.rPosition, percentBar2 := gUI.DiG5.D09Q2.rPercent, nameStr3 := gUI.DiG5.D10Q1.strName, posVal3 := gUI.DiG5.D10Q1.rPosition, percentBar3 := gUI.DiG5.D10Q1.rPercent, nameStr4 := gUI.DiG5.D10Q2.strName, posVal4 := gUI.DiG5.D10Q2.rPosition, percentBar4 := gUI.DiG5.D10Q2.rPercent, nameStr5 := gUI.DiG5.D11Q1.strName, posVal5 := gUI.DiG5.D11Q1.rPosition, percentBar5 := gUI.DiG5.D11Q1.rPercent, nameStr6 := gUI.DiG5.D11Q2.strName, posVal6 := gUI.DiG5.D11Q2.rPosition, percentBar6 := gUI.DiG5.D11Q2.rPercent, nameStr7 := gUI.DiG5.D12Q1.strName, posVal7 := gUI.DiG5.D12Q1.rPosition, percentBar7 := gUI.DiG5.D12Q1.rPercent, nameStr8 := gUI.DiG5.D12Q2.strName, posVal8 := gUI.DiG5.D12Q2.rPosition, percentBar8 := gUI.DiG5.D12Q2.rPercent)
    Frame (918,31 261x106)
        shows ModuleDTD(enable := gUI.DiG3.bRVD3_enable, propPercent := gUI.DiG3.rRVD3Percent)
    Frame (918,201 261x106)
        shows ModuleDTD(enable := gUI.DiG4.bRVD4_enable, propPercent := gUI.DiG5.rRVD5Percent)
    Frame (918,371 261x106)
        shows ModuleDTD(enable := gUI.DiG5.bRVD5_enable, propPercent := gUI.DiG5.rRVD5Percent)
    Line (10,175) (1250,175)
    Line (10,345) (1250,345)
END_VISUALIZATION

// Device/Application/display/Orig/Floor_Rail6
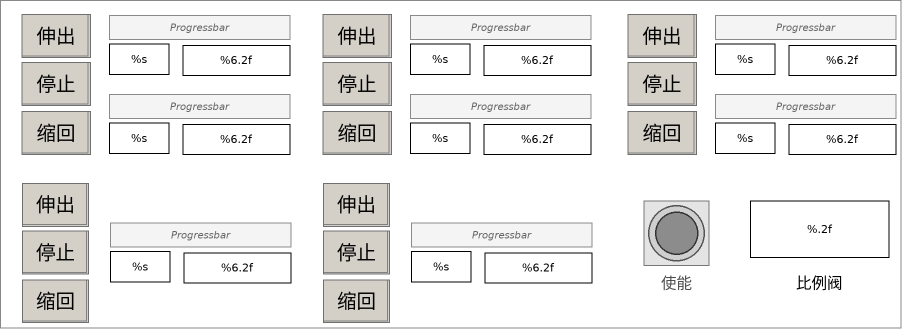
VISUALIZATION Floor_Rail6  // 902x329
    Frame (2,169 293x158)
        shows ModuleX1(extendButton := gUI.DiG6.S2.bExtend, retractButton := gUI.DiG6.S2.bRetract, stopButton := gUI.DiG6.S2.bStop, nameStr := gUI.DiG6.D15Q.strName, posVal := gUI.DiG6.D15Q.rPosition, percentBar := gUI.DiG6.D15Q.rPercent)
    Frame (2,3 292x156)
        shows ModuleX2(extendButton := gUI.DiG6.S1.bExtend, retractButton := gUI.DiG6.S1.bRetract, stopButton := gUI.DiG6.S1.bStop, nameStr1 := gUI.DiG6.D13Q.strName, posVal1 := gUI.DiG6.D13Q.rPosition, percentBar1 := gUI.DiG6.D13Q.rPercent, nameStr2 := gUI.DiG6.D14Q.strName, posVal2 := gUI.DiG6.D14Q.rPosition, percentBar2 := gUI.DiG6.D14Q.rPercent)
    Frame (303,3 292x156)
        shows ModuleX2(extendButton := gUI.DiG6.S1.bExtend, retractButton := gUI.DiG6.S1.bRetract, stopButton := gUI.DiG6.S1.bStop, nameStr1 := gUI.DiG6.D13L.strName, posVal1 := gUI.DiG6.D13L.rPosition, percentBar1 := gUI.DiG6.D13L.rPercent, nameStr2 := gUI.DiG6.D14L.strName, posVal2 := gUI.DiG6.D14L.rPosition, percentBar2 := gUI.DiG6.D14L.rPercent)
    Frame (303,169 293x158)
        shows ModuleX1(extendButton := gUI.DiG6.S4.bExtend, retractButton := gUI.DiG6.S4.bRetract, stopButton := gUI.DiG6.S4.bStop, nameStr := gUI.DiG6.D15L.strName, posVal := gUI.DiG6.D15L.rPosition, percentBar := gUI.DiG6.D15L.rPercent)
    Frame (608,3 292x156)
        shows ModuleX2(extendButton := gUI.DiG6.S5.bExtend, retractButton := gUI.DiG6.S5.bRetract, stopButton := gUI.DiG6.S5.bStop, nameStr1 := gUI.DiG6.D16L1.strName, posVal1 := gUI.DiG6.D16L1.rPosition, percentBar1 := gUI.DiG6.D16L1.rPercent, nameStr2 := gUI.DiG6.D16L2.strName, posVal2 := gUI.DiG6.D16L2.rPosition, percentBar2 := gUI.DiG6.D16L2.rPercent)
    Frame (630,195 261x106)
        shows ModuleDTD(enable := gUI.DiG6.bRVD6_enable, propPercent := gUI.DiG6.rRVD6Percent)
END_VISUALIZATION

// Device/Application/display/Orig/Floor_Rail7
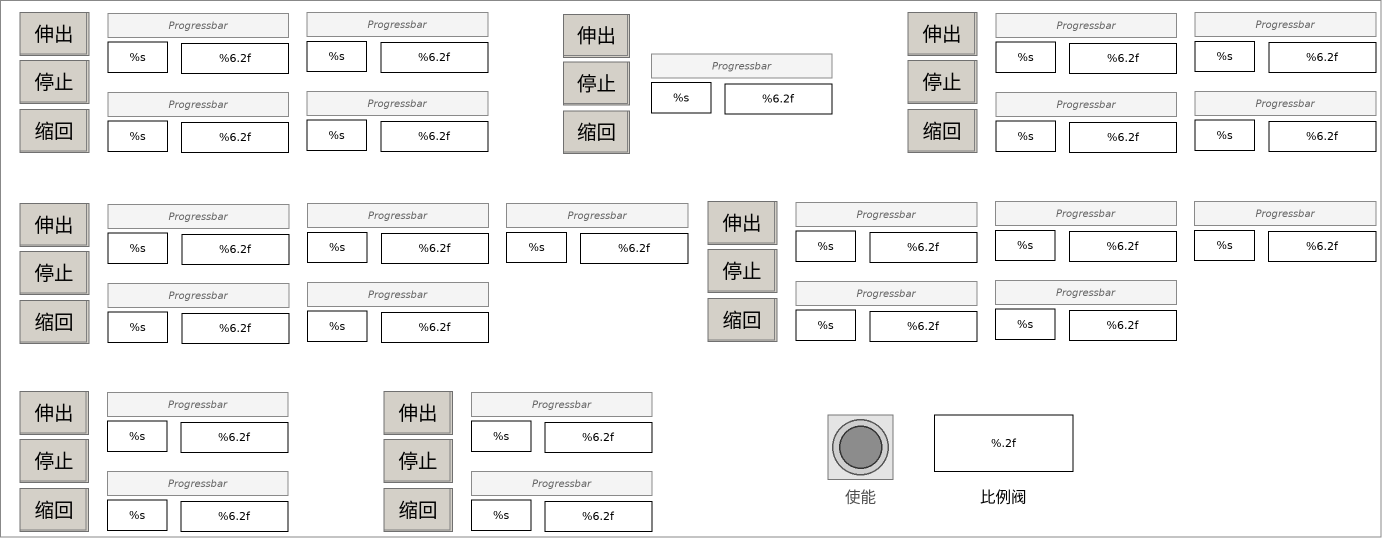
VISUALIZATION Floor_Rail7  // 1382x538
    Frame (0,1 492x156)
        shows ModuleX4(extendButton := gUI.DiG7.S1.bExtend, retractButton := gUI.DiG7.S1.bRetract, stopButton := gUI.DiG7.S1.bStop, nameStr1 := gUI.DiG7.D18L.strName, posVal1 := gUI.DiG7.D18L.rPosition, percentBar1 := gUI.DiG7.D18L.rPercent, nameStr2 := gUI.DiG7.D19L.strName, posVal2 := gUI.DiG7.D19L.rPosition, percentBar2 := gUI.DiG7.D19L.rPercent, nameStr3 := gUI.DiG7.D20L.strName, posVal3 := gUI.DiG7.D20L.rPosition, percentBar3 := gUI.DiG7.D20L.rPercent, nameStr4 := gUI.DiG7.D21L.strName, posVal4 := gUI.DiG7.D21L.rPosition, percentBar4 := gUI.DiG7.D21L.rPercent)
    Frame (543,0 293x158)
        shows ModuleX1(extendButton := gUI.DiG7.S2.bExtend, retractButton := gUI.DiG7.S2.bRetract, stopButton := gUI.DiG7.S2.bStop, nameStr := gUI.DiG7.D22L.strName, posVal := gUI.DiG7.D22L.rPosition, percentBar := gUI.DiG7.D22L.rPercent)
    Frame (888,1 492x156)
        shows ModuleX4(extendButton := gUI.DiG7.S3.bExtend, retractButton := gUI.DiG7.S3.bRetract, stopButton := gUI.DiG7.S3.bStop, nameStr1 := gUI.DiG7.D23L.strName, posVal1 := gUI.DiG7.D23L.rPosition, percentBar1 := gUI.DiG7.D23L.rPercent, nameStr2 := gUI.DiG7.D24L.strName, posVal2 := gUI.DiG7.D24L.rPosition, percentBar2 := gUI.DiG7.D24L.rPercent, nameStr3 := gUI.DiG7.D25L.strName, posVal3 := gUI.DiG7.D25L.rPosition, percentBar3 := gUI.DiG7.D25L.rPercent, nameStr4 := gUI.DiG7.D26L.strName, posVal4 := gUI.DiG7.D26L.rPosition, percentBar4 := gUI.DiG7.D26L.rPercent)
    Frame (0,192 692x156)
        shows ModuleX5(extendButton := gUI.DiG7.S4.bExtend, retractButton := gUI.DiG7.S4.bRetract, stopButton := gUI.DiG7.S4.bStop, nameStr1 := gUI.DiG7.D17Q.strName, posVal1 := gUI.DiG7.D17Q.rPosition, percentBar1 := gUI.DiG7.D17Q.rPercent, nameStr2 := gUI.DiG7.D18Q.strName, posVal2 := gUI.DiG7.D18Q.rPosition, percentBar2 := gUI.DiG7.D18Q.rPercent, nameStr3 := gUI.DiG7.D19Q.strName, posVal3 := gUI.DiG7.D19Q.rPosition, percentBar3 := gUI.DiG7.D19Q.rPercent, nameStr4 := gUI.DiG7.D20Q.strName, posVal4 := gUI.DiG7.D20Q.rPosition, percentBar4 := gUI.DiG7.D20Q.rPercent, nameStr5 := gUI.DiG7.D21Q.strName, posVal5 := gUI.DiG7.D21Q.rPosition, percentBar5 := gUI.DiG7.D21Q.rPercent)
    Frame (688,190 692x156)
        shows ModuleX5(extendButton := gUI.DiG7.S5.bExtend, retractButton := gUI.DiG7.S5.bRetract, stopButton := gUI.DiG7.S5.bStop, nameStr1 := gUI.DiG7.D22Q.strName, posVal1 := gUI.DiG7.D22Q.rPosition, percentBar1 := gUI.DiG7.D22Q.rPercent, nameStr2 := gUI.DiG7.D23Q.strName, posVal2 := gUI.DiG7.D23Q.rPosition, percentBar2 := gUI.DiG7.D23Q.rPercent, nameStr3 := gUI.DiG7.D24Q.strName, posVal3 := gUI.DiG7.D24Q.rPosition, percentBar3 := gUI.DiG7.D24Q.rPercent, nameStr4 := gUI.DiG7.D25Q.strName, posVal4 := gUI.DiG7.D25Q.rPosition, percentBar4 := gUI.DiG7.D25Q.rPercent, nameStr5 := gUI.DiG7.D26Q.strName, posVal5 := gUI.DiG7.D26Q.rPosition, percentBar5 := gUI.DiG7.D26Q.rPercent)
    Frame (0,380 292x156)
        shows ModuleX2(extendButton := gUI.DiG7.S6.bExtend, retractButton := gUI.DiG7.S6.bRetract, stopButton := gUI.DiG7.S6.bStop, nameStr1 := gUI.DiG7.D17L1.strName, posVal1 := gUI.DiG7.D17L1.rPosition, percentBar1 := gUI.DiG7.D17L1.rPercent, nameStr2 := gUI.DiG7.D17L2.strName, posVal2 := gUI.DiG7.D17L2.rPosition, percentBar2 := gUI.DiG7.D17L2.rPercent)
    Frame (364,380 292x156)
        shows ModuleX2(extendButton := gUI.DiG7.S7.bExtend, retractButton := gUI.DiG7.S7.bRetract, stopButton := gUI.DiG7.S7.bStop, nameStr1 := gUI.DiG7.D27L1.strName, posVal1 := gUI.DiG7.D27L1.rPosition, percentBar1 := gUI.DiG7.D27L1.rPercent, nameStr2 := gUI.DiG7.D27L2.strName, posVal2 := gUI.DiG7.D27L2.rPosition, percentBar2 := gUI.DiG7.D27L2.rPercent)
    Frame (814,409 261x106)
        shows ModuleDTD(enable := gUI.DiG7.bRVD7_enable, propPercent := gUI.DiG7.rRVD7Percent)
END_VISUALIZATION

// Device/Application/display/Floor_Rail
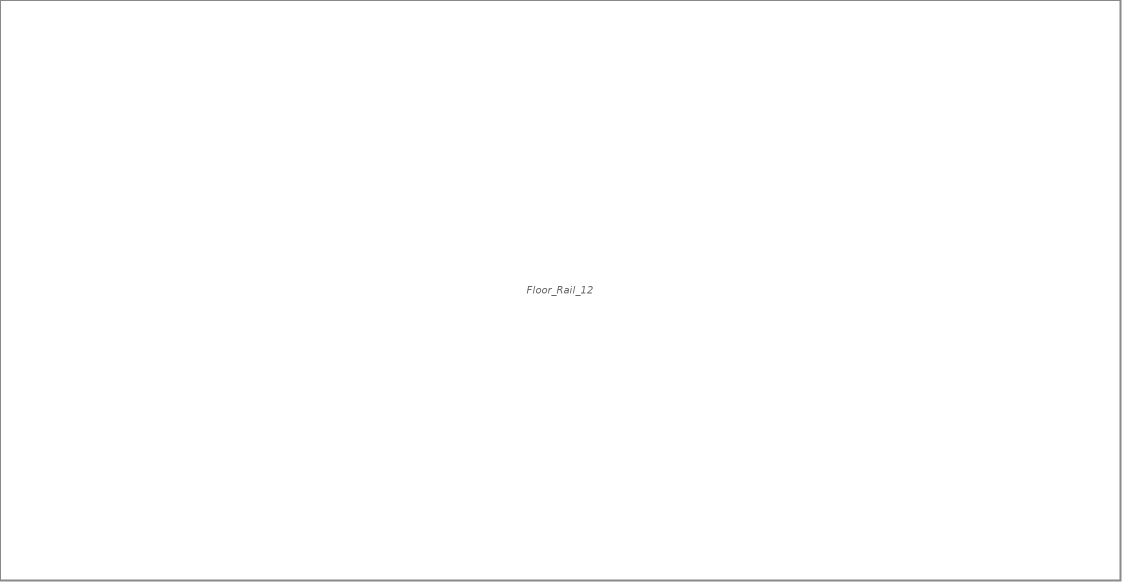
VISUALIZATION Floor_Rail  // 1122x582
    TabControl (0,0 1120x580)
        shows Floor_Rail_12()
        shows Floor_Rail_345()
        shows Floor_Rail6()
        shows Floor_Rail7()
        [0]: TabTitle=地轨p1-2, ImageId=__VisualizationStyle.Element-Clock-Blue
        [1]: TabTitle=地轨p3-5, ImageId=__VisualizationStyle.Element-Clock-Blue
        [2]: TabTitle=地轨p6, ImageId=__VisualizationStyle.Element-Clock-Blue
        [3]: TabTitle=地轨p7, ImageId=__VisualizationStyle.Element-Clock-Blue
END_VISUALIZATION

// Device/Application/display/Orig/Floor_Rail_12
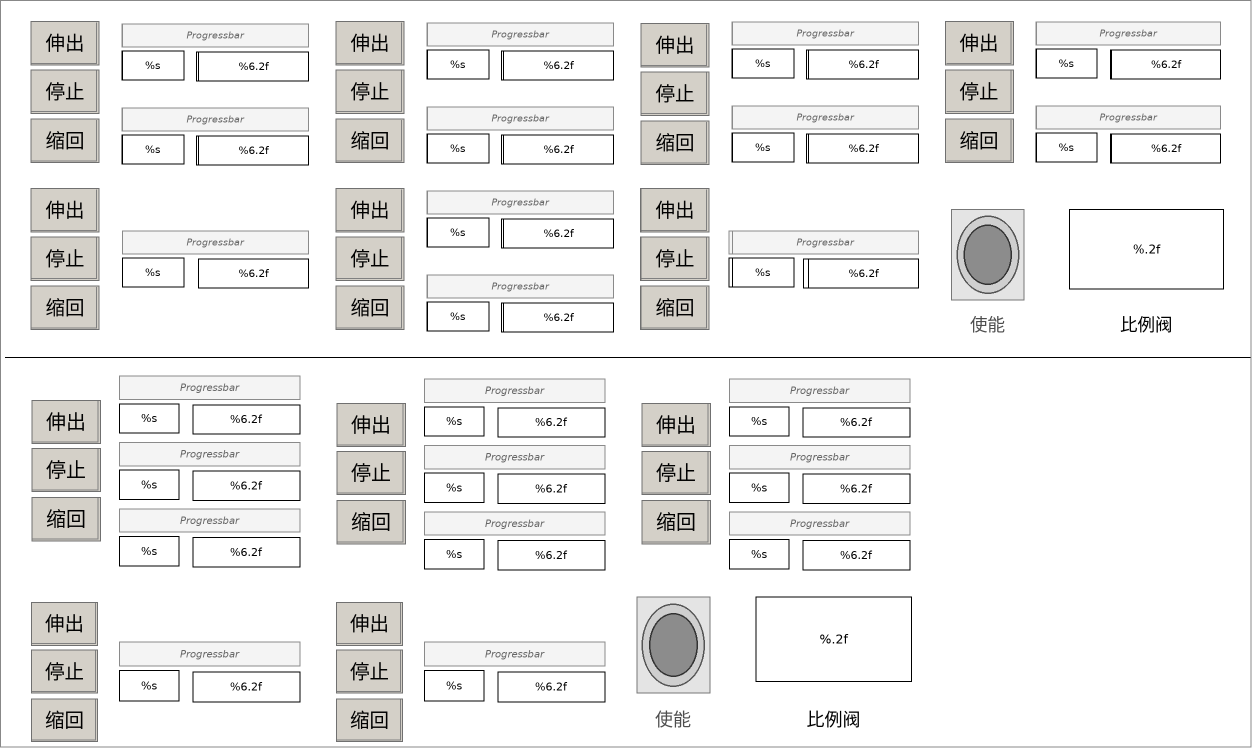
VISUALIZATION Floor_Rail_12  // 1252x748
    Group (18,16 1208x334)
        Group (305,0 293x150)
            Group (98,1 195x149)
                Frame (0,0 190x65)
                    shows OilBlock_PrimInfo(nameStr := gUI.DiG1.D28L1.strName, posVal := gUI.DiG1.D28L1.rPosition, percentBar := gUI.DiG1.D28L1.rPercent)
                Frame (0,84 190x65)
                    shows OilBlock_PrimInfo(nameStr := gUI.DiG1.D28L2.strName, posVal := gUI.DiG1.D28L2.rPosition, percentBar := gUI.DiG1.D28L2.rPercent)
            Frame (0,0 84x149)
                shows OilBlock_PrimButton(extendButton := gUI.DiG1.S2.bExtend, retractButton := gUI.DiG1.S2.bRetract, stopButton := gUI.DiG1.S2.bStop)
        Group (403,1 195x149)
            Frame (0,0 195x65)
                shows OilBlock_PrimInfo(nameStr := gUI.DiG1.D28L1.strName, posVal := gUI.DiG1.D28L1.rPosition, percentBar := gUI.DiG1.D28L1.rPercent)
            Frame (0,84 195x65)
                shows OilBlock_PrimInfo(nameStr := gUI.DiG1.D28L2.strName, posVal := gUI.DiG1.D28L2.rPosition, percentBar := gUI.DiG1.D28L2.rPercent)
        Frame (403,1 195x65)
            shows OilBlock_PrimInfo(nameStr := gUI.DiG1.D28L1.strName, posVal := gUI.DiG1.D28L1.rPosition, percentBar := gUI.DiG1.D28L1.rPercent)
        Frame (403,85 195x65)
            shows OilBlock_PrimInfo(nameStr := gUI.DiG1.D28L2.strName, posVal := gUI.DiG1.D28L2.rPosition, percentBar := gUI.DiG1.D28L2.rPercent)
        Frame (305,0 84x149)
            shows OilBlock_PrimButton(extendButton := gUI.DiG1.S2.bExtend, retractButton := gUI.DiG1.S2.bRetract, stopButton := gUI.DiG1.S2.bStop)
        Group (0,0 293x151)
            Frame (0,0 84x149)
                shows OilBlock_PrimButton(extendButton := gUI.DiG1.S1.bExtend, retractButton := gUI.DiG1.S1.bRetract, stopButton := gUI.DiG1.S1.bStop)
            Group (98,2 195x149)
                Frame (0,0 190x65)
                    shows OilBlock_PrimInfo(nameStr := gUI.DiG1.D00Q1.strName, posVal := gUI.DiG1.D00Q1.rPosition, percentBar := gUI.DiG1.D00Q1.rPercent)
                Frame (0,84 190x65)
                    shows OilBlock_PrimInfo(nameStr := gUI.DiG1.D00Q2.strName, posVal := gUI.DiG1.D00Q2.rPosition, percentBar := gUI.DiG1.D00Q2.rPercent)
        Frame (0,0 84x149)
            shows OilBlock_PrimButton(extendButton := gUI.DiG1.S1.bExtend, retractButton := gUI.DiG1.S1.bRetract, stopButton := gUI.DiG1.S1.bStop)
        Group (98,2 195x149)
            Frame (0,0 195x65)
                shows OilBlock_PrimInfo(nameStr := gUI.DiG1.D00Q1.strName, posVal := gUI.DiG1.D00Q1.rPosition, percentBar := gUI.DiG1.D00Q1.rPercent)
            Frame (0,84 195x65)
                shows OilBlock_PrimInfo(nameStr := gUI.DiG1.D00Q2.strName, posVal := gUI.DiG1.D00Q2.rPosition, percentBar := gUI.DiG1.D00Q2.rPercent)
        Frame (98,2 195x65)
            shows OilBlock_PrimInfo(nameStr := gUI.DiG1.D00Q1.strName, posVal := gUI.DiG1.D00Q1.rPosition, percentBar := gUI.DiG1.D00Q1.rPercent)
        Frame (98,86 195x65)
            shows OilBlock_PrimInfo(nameStr := gUI.DiG1.D00Q2.strName, posVal := gUI.DiG1.D00Q2.rPosition, percentBar := gUI.DiG1.D00Q2.rPercent)
        Group (0,167 293x149)
            Frame (98,42 195x65)
                shows OilBlock_PrimInfo(nameStr := gUI.DiG1.D01L.strName, posVal := gUI.DiG1.D01L.rPosition, percentBar := gUI.DiG1.D01L.rPercent)
            Frame (0,0 84x149)
                shows OilBlock_PrimButton(extendButton := gUI.DiG1.S5.bExtend, retractButton := gUI.DiG1.S5.bRetract, stopButton := gUI.DiG1.S5.bStop)
        Frame (98,209 195x65)
            shows OilBlock_PrimInfo(nameStr := gUI.DiG1.D01L.strName, posVal := gUI.DiG1.D01L.rPosition, percentBar := gUI.DiG1.D01L.rPercent)
        Frame (0,167 84x149)
            shows OilBlock_PrimButton(extendButton := gUI.DiG1.S5.bExtend, retractButton := gUI.DiG1.S5.bRetract, stopButton := gUI.DiG1.S5.bStop)
        Group (305,167 293x151)
            Group (98,2 195x149)
                Frame (0,0 190x65)
                    shows OilBlock_PrimInfo(nameStr := gUI.DiG1.D28Q.strName, posVal := gUI.DiG1.D28Q.rPosition, percentBar := gUI.DiG1.D28Q.rPercent)
                Frame (0,84 190x65)
                    shows OilBlock_PrimInfo(nameStr := gUI.DiG1.D29Q.strName, posVal := gUI.DiG1.D29Q.rPosition, percentBar := gUI.DiG1.D29Q.rPercent)
            Frame (0,0 84x149)
                shows OilBlock_PrimButton(extendButton := gUI.DiG1.S6.bExtend, retractButton := gUI.DiG1.S6.bRetract, stopButton := gUI.DiG1.S6.bStop)
        Group (403,169 195x149)
            Frame (0,0 195x65)
                shows OilBlock_PrimInfo(nameStr := gUI.DiG1.D28Q.strName, posVal := gUI.DiG1.D28Q.rPosition, percentBar := gUI.DiG1.D28Q.rPercent)
            Frame (0,84 195x65)
                shows OilBlock_PrimInfo(nameStr := gUI.DiG1.D29Q.strName, posVal := gUI.DiG1.D29Q.rPosition, percentBar := gUI.DiG1.D29Q.rPercent)
        Frame (403,169 195x65)
            shows OilBlock_PrimInfo(nameStr := gUI.DiG1.D28Q.strName, posVal := gUI.DiG1.D28Q.rPosition, percentBar := gUI.DiG1.D28Q.rPercent)
        Frame (403,253 195x65)
            shows OilBlock_PrimInfo(nameStr := gUI.DiG1.D29Q.strName, posVal := gUI.DiG1.D29Q.rPosition, percentBar := gUI.DiG1.D29Q.rPercent)
        Frame (305,167 84x149)
            shows OilBlock_PrimButton(extendButton := gUI.DiG1.S6.bExtend, retractButton := gUI.DiG1.S6.bRetract, stopButton := gUI.DiG1.S6.bStop)
        Group (610,0 293x151)
            Group (98,0 195x149)
                Frame (0,0 190x65)
                    shows OilBlock_PrimInfo(nameStr := gUI.DiG1.D29L.strName, posVal := gUI.DiG1.D29L.rPosition, percentBar := gUI.DiG1.D29L.rPercent)
                Frame (0,84 190x65)
                    shows OilBlock_PrimInfo(nameStr := gUI.DiG1.D30L.strName, posVal := gUI.DiG1.D30L.rPosition, percentBar := gUI.DiG1.D30L.rPercent)
            Frame (0,2 84x149)
                shows OilBlock_PrimButton(extendButton := gUI.DiG1.S3.bExtend, retractButton := gUI.DiG1.S3.bRetract, stopButton := gUI.DiG1.S3.bStop)
        Group (708,0 195x149)
            Frame (0,0 195x65)
                shows OilBlock_PrimInfo(nameStr := gUI.DiG1.D29L.strName, posVal := gUI.DiG1.D29L.rPosition, percentBar := gUI.DiG1.D29L.rPercent)
            Frame (0,84 195x65)
                shows OilBlock_PrimInfo(nameStr := gUI.DiG1.D30L.strName, posVal := gUI.DiG1.D30L.rPosition, percentBar := gUI.DiG1.D30L.rPercent)
        Frame (708,0 195x65)
            shows OilBlock_PrimInfo(nameStr := gUI.DiG1.D29L.strName, posVal := gUI.DiG1.D29L.rPosition, percentBar := gUI.DiG1.D29L.rPercent)
        Frame (708,84 195x65)
            shows OilBlock_PrimInfo(nameStr := gUI.DiG1.D30L.strName, posVal := gUI.DiG1.D30L.rPosition, percentBar := gUI.DiG1.D30L.rPercent)
        Frame (610,2 84x149)
            shows OilBlock_PrimButton(extendButton := gUI.DiG1.S3.bExtend, retractButton := gUI.DiG1.S3.bRetract, stopButton := gUI.DiG1.S3.bStop)
        Group (610,167 293x149)
            Group (0,0 293x149)
                Frame (95,42 190x65)
                    shows OilBlock_PrimInfo(nameStr := gUI.DiG1.D30Q.strName, posVal := gUI.DiG1.D30Q.rPosition, percentBar := gUI.DiG1.D30Q.rPercent)
                Frame (0,0 82x149)
                    shows OilBlock_PrimButton(extendButton := gUI.DiG1.S7.bExtend, retractButton := gUI.DiG1.S7.bRetract, stopButton := gUI.DiG1.S7.bStop)
            Frame (98,42 195x65)
                shows OilBlock_PrimInfo(nameStr := gUI.DiG1.D30Q.strName, posVal := gUI.DiG1.D30Q.rPosition, percentBar := gUI.DiG1.D30Q.rPercent)
            Frame (0,0 84x149)
                shows OilBlock_PrimButton(extendButton := gUI.DiG1.S7.bExtend, retractButton := gUI.DiG1.S7.bRetract, stopButton := gUI.DiG1.S7.bStop)
        Group (915,0 290x149)
            Group (97,0 193x149)
                Frame (0,0 190x65)
                    shows OilBlock_PrimInfo(nameStr := gUI.DiG1.D00L1.strName, posVal := gUI.DiG1.D00L1.rPosition, percentBar := gUI.DiG1.D00L1.rPercent)
                Frame (0,84 190x65)
                    shows OilBlock_PrimInfo(nameStr := gUI.DiG1.D00L2.strName, posVal := gUI.DiG1.D00L2.rPosition, percentBar := gUI.DiG1.D00L2.rPercent)
            Frame (0,0 83x149)
                shows OilBlock_PrimButton(extendButton := gUI.DiG1.S4.bExtend, retractButton := gUI.DiG1.S4.bRetract, stopButton := gUI.DiG1.S4.bStop)
        Group (1012,0 193x149)
            Frame (0,0 193x65)
                shows OilBlock_PrimInfo(nameStr := gUI.DiG1.D00L1.strName, posVal := gUI.DiG1.D00L1.rPosition, percentBar := gUI.DiG1.D00L1.rPercent)
            Frame (0,84 193x65)
                shows OilBlock_PrimInfo(nameStr := gUI.DiG1.D00L2.strName, posVal := gUI.DiG1.D00L2.rPosition, percentBar := gUI.DiG1.D00L2.rPercent)
        Frame (1012,0 193x65)
            shows OilBlock_PrimInfo(nameStr := gUI.DiG1.D00L1.strName, posVal := gUI.DiG1.D00L1.rPosition, percentBar := gUI.DiG1.D00L1.rPercent)
        Frame (1012,84 193x65)
            shows OilBlock_PrimInfo(nameStr := gUI.DiG1.D00L2.strName, posVal := gUI.DiG1.D00L2.rPosition, percentBar := gUI.DiG1.D00L2.rPercent)
        Frame (915,0 83x149)
            shows OilBlock_PrimButton(extendButton := gUI.DiG1.S4.bExtend, retractButton := gUI.DiG1.S4.bRetract, stopButton := gUI.DiG1.S4.bStop)
        Frame (918,185 290x149)
            shows ModuleDTD(enable := gUI.DiG1.bRVD1_enable, propPercent := gUI.DiG1.rRVD1Percent)
    Group (11,364 903x382)
        Frame (0,0 293x207)
            shows ModuleX3(extendButton := gUI.DiG2.S1.bExtend, retractButton := gUI.DiG2.S1.bRetract, stopButton := gUI.DiG2.S1.bStop, nameStr1 := gUI.DiG2.D02L.strName, posVal1 := gUI.DiG2.D02L.rPosition, percentBar1 := gUI.DiG2.D02L.rPercent, nameStr2 := gUI.DiG2.D03L.strName, posVal2 := gUI.DiG2.D03L.rPosition, percentBar2 := gUI.DiG2.D03L.rPercent, nameStr3 := gUI.DiG2.D04L.strName, posVal3 := gUI.DiG2.D04L.rPosition, percentBar3 := gUI.DiG2.D04L.rPercent)
        Frame (0,224 293x158)
            shows ModuleX1(extendButton := gUI.DiG2.S2.bExtend, retractButton := gUI.DiG2.S2.bRetract, stopButton := gUI.DiG2.S2.bStop, nameStr := gUI.DiG2.D05L.strName, posVal := gUI.DiG2.D05L.rPosition, percentBar := gUI.DiG2.D05L.rPercent)
        Frame (305,3 293x207)
            shows ModuleX3(extendButton := gUI.DiG2.S3.bExtend, retractButton := gUI.DiG2.S3.bRetract, stopButton := gUI.DiG2.S3.bStop, nameStr1 := gUI.DiG2.D06L.strName, posVal1 := gUI.DiG2.D06L.rPosition, percentBar1 := gUI.DiG2.D06L.rPercent, nameStr2 := gUI.DiG2.D07L.strName, posVal2 := gUI.DiG2.D07L.rPosition, percentBar2 := gUI.DiG2.D07L.rPercent, nameStr3 := gUI.DiG2.D08L.strName, posVal3 := gUI.DiG2.D08L.rPosition, percentBar3 := gUI.DiG2.D08L.rPercent)
        Frame (305,224 293x158)
            shows ModuleX1(extendButton := gUI.DiG2.S4.bExtend, retractButton := gUI.DiG2.S4.bRetract, stopButton := gUI.DiG2.S4.bStop, nameStr := gUI.DiG2.D09L.strName, posVal := gUI.DiG2.D09L.rPosition, percentBar := gUI.DiG2.D09L.rPercent)
        Frame (610,3 293x207)
            shows ModuleX3(extendButton := gUI.DiG2.S5.bExtend, retractButton := gUI.DiG2.S5.bRetract, stopButton := gUI.DiG2.S5.bStop, nameStr1 := gUI.DiG2.D10L.strName, posVal1 := gUI.DiG2.D10L.rPosition, percentBar1 := gUI.DiG2.D10L.rPercent, nameStr2 := gUI.DiG2.D11L.strName, posVal2 := gUI.DiG2.D11L.rPosition, percentBar2 := gUI.DiG2.D11L.rPercent, nameStr3 := gUI.DiG2.D12L.strName, posVal3 := gUI.DiG2.D12L.rPosition, percentBar3 := gUI.DiG2.D12L.rPercent)
        Frame (610,224 293x158)
            shows ModuleDTD(enable := gUI.DiG2.bRVD2_enable, propPercent := gUI.DiG2.rRVD2Percent)
    Line (5,357) (1250,357)
END_VISUALIZATION

// Device/Application/display/main_UI
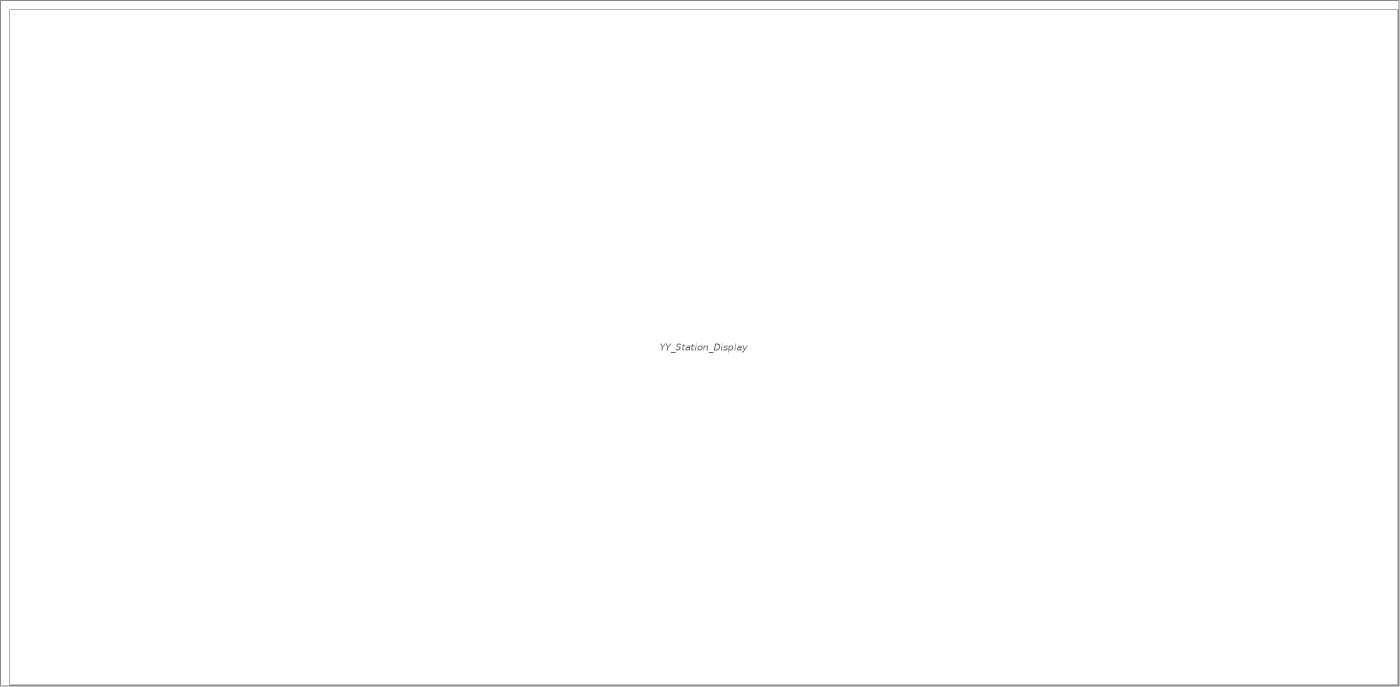
VISUALIZATION main_UI  // 1509x741
    TabControl (10,10 1497x729)
        shows YY_Station_Display()
        shows Floor_Rail()
        [0]: TabTitle=液压站
        [1]: TabTitle=地轨
END_VISUALIZATION

(* text list TextList (id | default)
  1 | 2
  2 | 3
   |  *)
